LIN {X 0,Y 420.626,Z 325.953,A -85,B 0,C 180,E1 -10192.084,E2 -10192.084} C_VEL
LIN {X 0,Y 421.329,Z 314.236,A -85,B 0,C 180,E1 -10194.385,E2 -10194.385} C_VEL
LIN {X 0,Y 419.422,Z 303.683,A -85,B 0,C 180,E1 -10196.632,E2 -10196.632} C_VEL
LIN {X 0,Y 418.338,Z 298.378,A -85,B 0,C 180,E1 -10197.821,E2 -10197.821} C_VEL
LIN {X 0,Y 418.216,Z 298.389,A -85,B 0,C 180,E1 -10201.397,E2 -10201.397} C_VEL
LIN {X 0,Y 418.27,Z 298.382,A -85,B 0,C 180,E1 -10204.581,E2 -10204.581} C_VEL
LIN {X 0,Y 418.228,Z 298.387,A -85,B 0,C 180,E1 -10207.833,E2 -10207.833} C_VEL
LIN {X 0,Y 418.225,Z 298.385,A -85,B 0,C 180,E1 -10210.948,E2 -10210.948} C_VEL
LIN {X 0,Y 418.211,Z 298.387,A -85,B 0,C 180,E1 -10213.729,E2 -10213.729} C_VEL
LIN {X 0,Y 418.211,Z 298.394,A -85,B 0,C 180,E1 -10216.449,E2 -10216.449} C_VEL
LIN {X 0,Y 418.224,Z 298.386,A -85,B 0,C 180,E1 -10219.13,E2 -10219.13} C_VEL
LIN {X 0,Y 418.228,Z 298.387,A -85,B 0,C 180,E1 -10222.167,E2 -10222.167} C_VEL
LIN {X 0,Y 418.264,Z 298.38,A -85,B 0,C 180,E1 -10225.42,E2 -10225.42} C_VEL
LIN {X 0,Y 418.21,Z 298.392,A -85,B 0,C 180,E1 -10228.604,E2 -10228.604} C_VEL
LIN {X 0,Y 418.288,Z 298.376,A -85,B 0,C 180,E1 -10231.936,E2 -10231.936} C_VEL
LIN {X 0,Y 418.288,Z 298.381,A -85,B 0,C 180,E1 -10235.162,E2 -10235.162} C_VEL
LIN {X 0,Y 418.229,Z 298.385,A -85,B 0,C 180,E1 -10238.303,E2 -10238.303} C_VEL
LIN {X 0,Y 418.277,Z 298.381,A -85,B 0,C 180,E1 -10241.383,E2 -10241.383} C_VEL
LIN {X 0,Y 418.295,Z 298.376,A -85,B 0,C 180,E1 -10244.406,E2 -10244.406} C_VEL
LIN {X 0,Y 418.349,Z 298.374,A -85,B 0,C 180,E1 -10247.385,E2 -10247.385} C_VEL
LIN {X 0,Y 418.394,Z 298.371,A -85,B 0,C 180,E1 -10251.305,E2 -10251.305} C_VEL
LIN {X 0,Y 418.483,Z 298.359,A -85,B 0,C 180,E1 -10253.249,E2 -10253.249} C_VEL
LIN {X 0,Y 418.326,Z 298.377,A -85,B 0,C 180,E1 -10255.181,E2 -10255.181} C_VEL
LIN {X 0,Y 418.532,Z 298.347,A -85,B 0,C 180,E1 -10258.075,E2 -10258.075} C_VEL
LIN {X 0,Y 418.658,Z 298.332,A -85,B 0,C 180,E1 -10260,E2 -10260} C_VEL
LIN {X 0,Y 418.49,Z 298.352,A -85,B 0,C 180,E1 -10262.888,E2 -10262.888} C_VEL
LIN {X 0,Y 418.438,Z 298.358,A -85,B 0,C 180,E1 -10266.529,E2 -10266.529} C_VEL
LIN {X 0,Y 418.331,Z 298.379,A -85,B 0,C 180,E1 -10269.672,E2 -10269.672} C_VEL
LIN {X 0,Y 418.34,Z 298.37,A -85,B 0,C 180,E1 -10273,E2 -10273} C_VEL
LIN {X 0,Y 418.306,Z 298.374,A -85,B 0,C 180,E1 -10276.734,E2 -10276.734} C_VEL
LIN {X 0,Y 418.265,Z 298.385,A -85,B 0,C 180,E1 -10279.79,E2 -10279.79} C_VEL
LIN {X 0,Y 418.222,Z 298.385,A -85,B 0,C 180,E1 -10282.737,E2 -10282.737} C_VEL
LIN {X 0,Y 418.213,Z 298.391,A -85,B 0,C 180,E1 -10285.908,E2 -10285.908} C_VEL
LIN {X 0,Y 418.254,Z 298.381,A -85,B 0,C 180,E1 -10289.163,E2 -10289.163} C_VEL
LIN {X 0,Y 418.238,Z 298.387,A -85,B 0,C 180,E1 -10292.529,E2 -10292.529} C_VEL
LIN {X 0,Y 418.247,Z 298.383,A -85,B 0,C 180,E1 -10294.842,E2 -10294.842} C_VEL
LIN {X 0,Y 418.225,Z 298.392,A -85,B 0,C 180,E1 -10298.445,E2 -10298.445} C_VEL
LIN {X 0,Y 418.206,Z 298.389,A -85,B 0,C 180,E1 -10300.95,E2 -10300.95} C_VEL
LIN {X 0,Y 418.191,Z 298.389,A -85,B 0,C 180,E1 -10303.726,E2 -10303.726} C_VEL
LIN {X 0,Y 418.179,Z 298.396,A -85,B 0,C 180,E1 -10306.444,E2 -10306.444} C_VEL
LIN {X 0,Y 418.207,Z 298.389,A -85,B 0,C 180,E1 -10309.133,E2 -10309.133} C_VEL
LIN {X 0,Y 418.225,Z 298.392,A -85,B 0,C 180,E1 -10312.773,E2 -10312.773} C_VEL
LIN {X 0,Y 418.197,Z 298.39,A -85,B 0,C 180,E1 -10316.317,E2 -10316.317} C_VEL
LIN {X 0,Y 418.237,Z 298.383,A -85,B 0,C 180,E1 -10319.726,E2 -10319.726} C_VEL
LIN {X 0,Y 418.201,Z 298.395,A -85,B 0,C 180,E1 -10323.014,E2 -10323.014} C_VEL
LIN {X 0,Y 418.26,Z 298.38,A -85,B 0,C 180,E1 -10326.216,E2 -10326.216} C_VEL
LIN {X 0,Y 418.255,Z 298.386,A -85,B 0,C 180,E1 -10329.335,E2 -10329.335} C_VEL
LIN {X 0,Y 418.283,Z 298.377,A -85,B 0,C 180,E1 -10332.394,E2 -10332.394} C_VEL
LIN {X 0,Y 418.3,Z 298.381,A -85,B 0,C 180,E1 -10335.401,E2 -10335.401} C_VEL
LIN {X 0,Y 418.316,Z 298.373,A -85,B 0,C 180,E1 -10338.367,E2 -10338.367} C_VEL
LIN {X 0,Y 418.451,Z 298.356,A -85,B 0,C 180,E1 -10342.276,E2 -10342.276} C_VEL
LIN {X 0,Y 418.474,Z 298.354,A -85,B 0,C 180,E1 -10344.214,E2 -10344.214} C_VEL
LIN {X 0,Y 418.536,Z 298.348,A -85,B 0,C 180,E1 -10348.072,E2 -10348.072} C_VEL
LIN {X 0,Y 418.545,Z 298.348,A -85,B 0,C 180,E1 -10349.997,E2 -10349.997} C_VEL
LIN {X 0,Y 418.474,Z 298.353,A -85,B 0,C 180,E1 -10352.885,E2 -10352.885} C_VEL
LIN {X 0,Y 418.484,Z 298.36,A -85,B 0,C 180,E1 -10355.78,E2 -10355.78} C_VEL
LIN {X 0,Y 418.36,Z 298.372,A -85,B 0,C 180,E1 -10359.132,E2 -10359.132} C_VEL
LIN {X 0,Y 418.401,Z 298.488,A -85,B 0,C 180,E1 -10359.758,E2 -10359.758} C_VEL
LIN {X 0,Y 420.017,Z 308.097,A -85,B 0,C 180,E1 -10362.069,E2 -10362.069} C_VEL
LIN {X 0,Y 419.967,Z 311.749,A -85,B 0,C 180,E1 -10362.899,E2 -10362.899} C_VEL
LIN {X 0,Y 419.417,Z 313.02,A -85,B 0,C 180,E1 -10363.037,E2 -10363.037} C_VEL
LIN {X 0,Y 417.673,Z 315.322,A -85,B 0,C 180,E1 -10363.058,E2 -10363.058} C_VEL
LIN {X 0,Y 411.938,Z 322.29,A -85,B 0,C 180,E1 -10362.926,E2 -10362.926} C_VEL
LIN {X 0,Y 410.732,Z 325.842,A -85,B 0,C 180,E1 -10362.932,E2 -10362.932} C_VEL
LIN {X 0,Y 411.108,Z 329.038,A -85,B 0,C 180,E1 -10362.976,E2 -10362.976} C_VEL
LIN {X 0,Y 412.467,Z 332.294,A -85,B 0,C 180,E1 -10363.092,E2 -10363.092} C_VEL
LIN {X 0,Y 416.345,Z 339.616,A -85,B 0,C 180,E1 -10363.438,E2 -10363.438} C_VEL
LIN {X 0,Y 416.967,Z 343.12,A -85,B 0,C 180,E1 -10363.539,E2 -10363.539} C_VEL
LIN {X 0,Y 415.843,Z 420.461,A -85,B 0,C 180,E1 -10364.928,E2 -10364.928} C_VEL
LIN {X 0,Y 415.479,Z 434.115,A -85,B 0,C 180,E1 -10365.381,E2 -10365.381} C_VEL
LIN {X 0,Y 414.977,Z 446.178,A -85,B 0,C 180,E1 -10365.97,E2 -10365.97} C_VEL
LIN {X 0,Y 414.346,Z 458.066,A -85,B 0,C 180,E1 -10366.755,E2 -10366.755} C_VEL
LIN {X 0,Y 413.671,Z 468.928,A -85,B 0,C 180,E1 -10367.674,E2 -10367.674} C_VEL
LIN {X 0,Y 412.901,Z 478.924,A -85,B 0,C 180,E1 -10368.722,E2 -10368.722} C_VEL
LIN {X 0,Y 412.298,Z 488.255,A -85,B 0,C 180,E1 -10369.928,E2 -10369.928} C_VEL
LIN {X 0,Y 411.669,Z 496.665,A -85,B 0,C 180,E1 -10371.266,E2 -10371.266} C_VEL
LIN {X 0,Y 411.078,Z 504.603,A -85,B 0,C 180,E1 -10372.838,E2 -10372.838} C_VEL
LIN {X 0,Y 410.701,Z 510.279,A -85,B 0,C 180,E1 -10374.243,E2 -10374.243} C_VEL
LIN {X 0,Y 410.361,Z 515.517,A -85,B 0,C 180,E1 -10375.89,E2 -10375.89} C_VEL
LIN {X 0,Y 410.1,Z 519.401,A -85,B 0,C 180,E1 -10377.556,E2 -10377.556} C_VEL
LIN {X 0,Y 409.937,Z 521.797,A -85,B 0,C 180,E1 -10379.032,E2 -10379.032} C_VEL
LIN {X 0,Y 409.815,Z 523.491,A -85,B 0,C 180,E1 -10380.956,E2 -10380.956} C_VEL
LIN {X 0,Y 409.824,Z 523.714,A -85,B 0,C 180,E1 -10382.829,E2 -10382.829} C_VEL
LIN {X 0,Y 409.879,Z 522.561,A -85,B 0,C 180,E1 -10384.61,E2 -10384.61} C_VEL
LIN {X 0,Y 410.105,Z 520.141,A -85,B 0,C 180,E1 -10386.347,E2 -10386.347} C_VEL
LIN {X 0,Y 410.345,Z 516.461,A -85,B 0,C 180,E1 -10388.059,E2 -10388.059} C_VEL
LIN {X 0,Y 410.695,Z 511.796,A -85,B 0,C 180,E1 -10389.64,E2 -10389.64} C_VEL
LIN {X 0,Y 411.086,Z 505.785,A -85,B 0,C 180,E1 -10391.216,E2 -10391.216} C_VEL
LIN {X 0,Y 411.689,Z 498.204,A -85,B 0,C 180,E1 -10392.772,E2 -10392.772} C_VEL
LIN {X 0,Y 412.444,Z 489.922,A -85,B 0,C 180,E1 -10394.139,E2 -10394.139} C_VEL
LIN {X 0,Y 413.206,Z 480.472,A -85,B 0,C 180,E1 -10395.408,E2 -10395.408} C_VEL
LIN {X 0,Y 413.948,Z 469.615,A -85,B 0,C 180,E1 -10396.573,E2 -10396.573} C_VEL
LIN {X 0,Y 414.77,Z 458.24,A -85,B 0,C 180,E1 -10397.54,E2 -10397.54} C_VEL
LIN {X 0,Y 415.403,Z 446.521,A -85,B 0,C 180,E1 -10398.315,E2 -10398.315} C_VEL
LIN {X 0,Y 415.954,Z 432.986,A -85,B 0,C 180,E1 -10398.966,E2 -10398.966} C_VEL
LIN {X 0,Y 416.385,Z 419.739,A -85,B 0,C 180,E1 -10399.384,E2 -10399.384} C_VEL
LIN {X 0,Y 417.604,Z 333.211,A -85,B 0,C 180,E1 -10400.949,E2 -10400.949} C_VEL
LIN {X 0,Y 413.3,Z 312.691,A -85,B 0,C 180,E1 -10401.573,E2 -10401.573} C_VEL
LIN {X 0,Y 413.042,Z 308.119,A -85,B 0,C 180,E1 -10402.534,E2 -10402.534} C_VEL
LIN {X 0,Y 411.183,Z 299.269,A -85,B 0,C 180,E1 -10404.52,E2 -10404.52} C_VEL
LIN {X 0,Y 411.127,Z 299.276,A -85,B 0,C 180,E1 -10407.999,E2 -10407.999} C_VEL
LIN {X 0,Y 411.181,Z 299.266,A -85,B 0,C 180,E1 -10411.407,E2 -10411.407} C_VEL
LIN {X 0,Y 411.195,Z 299.268,A -85,B 0,C 180,E1 -10413.616,E2 -10413.616} C_VEL
LIN {X 0,Y 411.158,Z 299.274,A -85,B 0,C 180,E1 -10416.85,E2 -10416.85} C_VEL
LIN {X 0,Y 411.167,Z 299.271,A -85,B 0,C 180,E1 -10420.049,E2 -10420.049} C_VEL
LIN {X 0,Y 411.216,Z 299.261,A -85,B 0,C 180,E1 -10423.129,E2 -10423.129} C_VEL
LIN {X 0,Y 411.256,Z 299.258,A -85,B 0,C 180,E1 -10426.895,E2 -10426.895} C_VEL
LIN {X 0,Y 411.242,Z 299.255,A -85,B 0,C 180,E1 -10430.16,E2 -10430.16} C_VEL
LIN {X 0,Y 411.407,Z 299.237,A -85,B 0,C 180,E1 -10433.132,E2 -10433.132} C_VEL
LIN {X 0,Y 411.259,Z 299.254,A -85,B 0,C 180,E1 -10435.098,E2 -10435.098} C_VEL
LIN {X 0,Y 411.463,Z 299.228,A -85,B 0,C 180,E1 -10438.042,E2 -10438.042} C_VEL
LIN {X 0,Y 411.59,Z 299.206,A -85,B 0,C 180,E1 -10440,E2 -10440} C_VEL
LIN {X 0,Y 411.422,Z 299.234,A -85,B 0,C 180,E1 -10442.937,E2 -10442.937} C_VEL
LIN {X 0,Y 411.41,Z 299.237,A -85,B 0,C 180,E1 -10446.868,E2 -10446.868} C_VEL
LIN {X 0,Y 411.262,Z 299.254,A -85,B 0,C 180,E1 -10449.84,E2 -10449.84} C_VEL
LIN {X 0,Y 411.265,Z 299.253,A -85,B 0,C 180,E1 -10453.11,E2 -10453.11} C_VEL
LIN {X 0,Y 411.217,Z 299.255,A -85,B 0,C 180,E1 -10456.871,E2 -10456.871} C_VEL
LIN {X 0,Y 411.21,Z 299.253,A -85,B 0,C 180,E1 -10459.988,E2 -10459.988} C_VEL
LIN {X 0,Y 411.18,Z 299.267,A -85,B 0,C 180,E1 -10463.149,E2 -10463.149} C_VEL
LIN {X 0,Y 411.197,Z 299.26,A -85,B 0,C 180,E1 -10466.384,E2 -10466.384} C_VEL
LIN {X 0,Y 411.169,Z 299.268,A -85,B 0,C 180,E1 -10469.715,E2 -10469.715} C_VEL
LIN {X 0,Y 411.168,Z 299.266,A -85,B 0,C 180,E1 -10473.159,E2 -10473.159} C_VEL
LIN {X 0,Y 411.165,Z 299.266,A -85,B 0,C 180,E1 -10476.558,E2 -10476.558} C_VEL
LIN {X 0,Y 411.204,Z 299.267,A -85,B 0,C 180,E1 -10479.736,E2 -10479.736} C_VEL
LIN {X 0,Y 411.2,Z 299.266,A -85,B 0,C 180,E1 -10483.13,E2 -10483.13} C_VEL
LIN {X 0,Y 411.208,Z 299.267,A -85,B 0,C 180,E1 -10485.876,E2 -10485.876} C_VEL
LIN {X 0,Y 411.188,Z 299.27,A -85,B 0,C 180,E1 -10489.504,E2 -10489.504} C_VEL
LIN {X 0,Y 411.182,Z 299.268,A -85,B 0,C 180,E1 -10492.032,E2 -10492.032} C_VEL
LIN {X 0,Y 411.186,Z 299.271,A -85,B 0,C 180,E1 -10495.671,E2 -10495.671} C_VEL
LIN {X 0,Y 411.18,Z 299.272,A -85,B 0,C 180,E1 -10499.158,E2 -10499.158} C_VEL
LIN {X 0,Y 411.278,Z 299.342,A -85,B 0,C 180,E1 -10502.115,E2 -10502.115} C_VEL
LIN {X 0,Y 413.936,Z 312.197,A -85,B 0,C 180,E1 -10504.889,E2 -10504.889} C_VEL
LIN {X 0,Y 414.359,Z 316.233,A -85,B 0,C 180,E1 -10505.718,E2 -10505.718} C_VEL
LIN {X 0,Y 413.189,Z 333.63,A -85,B 0,C 180,E1 -10509.077,E2 -10509.077} C_VEL
LIN {X 0,Y 412.799,Z 340.804,A -85,B 0,C 180,E1 -10510.452,E2 -10510.452} C_VEL
LIN {X 0,Y 417.216,Z 368.982,A -85,B 0,C 180,E1 -10511.211,E2 -10511.211} C_VEL
LIN {X 0,Y 416.076,Z 450.173,A -85,B 0,C 180,E1 -10512.685,E2 -10512.685} C_VEL
LIN {X 0,Y 415.495,Z 463.908,A -85,B 0,C 180,E1 -10513.135,E2 -10513.135} C_VEL
LIN {X 0,Y 414.854,Z 475.762,A -85,B 0,C 180,E1 -10513.709,E2 -10513.709} C_VEL
LIN {X 0,Y 414.048,Z 487.812,A -85,B 0,C 180,E1 -10514.498,E2 -10514.498} C_VEL
LIN {X 0,Y 413.318,Z 499.293,A -85,B 0,C 180,E1 -10515.475,E2 -10515.475} C_VEL
LIN {X 0,Y 412.495,Z 509.746,A -85,B 0,C 180,E1 -10516.581,E2 -10516.581} C_VEL
LIN {X 0,Y 411.872,Z 518.266,A -85,B 0,C 180,E1 -10517.689,E2 -10517.689} C_VEL
LIN {X 0,Y 411.086,Z 527.506,A -85,B 0,C 180,E1 -10519.165,E2 -10519.165} C_VEL
LIN {X 0,Y 410.621,Z 534.957,A -85,B 0,C 180,E1 -10520.646,E2 -10520.646} C_VEL
LIN {X 0,Y 410.284,Z 540.946,A -85,B 0,C 180,E1 -10522.127,E2 -10522.127} C_VEL
LIN {X 0,Y 410.056,Z 546.105,A -85,B 0,C 180,E1 -10523.759,E2 -10523.759} C_VEL
LIN {X 0,Y 410.017,Z 549.293,A -85,B 0,C 180,E1 -10525.087,E2 -10525.087} C_VEL
LIN {X 0,Y 409.932,Z 551.145,A -85,B 0,C 180,E1 -10526.071,E2 -10526.071} C_VEL
LIN {X 0,Y 409.996,Z 553.54,A -85,B 0,C 180,E1 -10528.039,E2 -10528.039} C_VEL
LIN {X 0,Y 409.955,Z 554.143,A -85,B 0,C 180,E1 -10529.021,E2 -10529.021} C_VEL
LIN {X 0,Y 409.949,Z 554.331,A -85,B 0,C 180,E1 -10530.003,E2 -10530.003} C_VEL
LIN {X 0,Y 409.997,Z 553.467,A -85,B 0,C 180,E1 -10531.968,E2 -10531.968} C_VEL
LIN {X 0,Y 409.932,Z 552.442,A -85,B 0,C 180,E1 -10532.951,E2 -10532.951} C_VEL
LIN {X 0,Y 409.935,Z 550.987,A -85,B 0,C 180,E1 -10533.935,E2 -10533.935} C_VEL
LIN {X 0,Y 410.018,Z 547.982,A -85,B 0,C 180,E1 -10535.412,E2 -10535.412} C_VEL
LIN {X 0,Y 410.167,Z 543.911,A -85,B 0,C 180,E1 -10536.891,E2 -10536.891} C_VEL
LIN {X 0,Y 410.458,Z 537.642,A -85,B 0,C 180,E1 -10538.619,E2 -10538.619} C_VEL
LIN {X 0,Y 410.845,Z 530.811,A -85,B 0,C 180,E1 -10540.101,E2 -10540.101} C_VEL
LIN {X 0,Y 411.441,Z 522.309,A -85,B 0,C 180,E1 -10541.581,E2 -10541.581} C_VEL
LIN {X 0,Y 412.06,Z 513.546,A -85,B 0,C 180,E1 -10542.813,E2 -10542.813} C_VEL
LIN {X 0,Y 412.801,Z 503.481,A -85,B 0,C 180,E1 -10543.967,E2 -10543.967} C_VEL
LIN {X 0,Y 413.548,Z 492.018,A -85,B 0,C 180,E1 -10545.023,E2 -10545.023} C_VEL
LIN {X 0,Y 414.325,Z 479.976,A -85,B 0,C 180,E1 -10545.876,E2 -10545.876} C_VEL
LIN {X 0,Y 414.998,Z 467.447,A -85,B 0,C 180,E1 -10546.544,E2 -10546.544} C_VEL
LIN {X 0,Y 415.559,Z 454.361,A -85,B 0,C 180,E1 -10547.027,E2 -10547.027} C_VEL
LIN {X 0,Y 415.931,Z 437.009,A -85,B 0,C 180,E1 -10547.392,E2 -10547.392} C_VEL
LIN {X 0,Y 416.689,Z 368.049,A -85,B 0,C 180,E1 -10548.617,E2 -10548.617} C_VEL
LIN {X 0,Y 412.668,Z 341.785,A -85,B 0,C 180,E1 -10549.281,E2 -10549.281} C_VEL
LIN {X 0,Y 413.701,Z 325.613,A -85,B 0,C 180,E1 -10552.474,E2 -10552.474} C_VEL
LIN {X 0,Y 414.371,Z 315.206,A -85,B 0,C 180,E1 -10554.555,E2 -10554.555} C_VEL
LIN {X 0,Y 412.159,Z 303.311,A -85,B 0,C 180,E1 -10557.139,E2 -10557.139} C_VEL
LIN {X 0,Y 411.278,Z 299.257,A -85,B 0,C 180,E1 -10558.1,E2 -10558.1} C_VEL
LIN {X 0,Y 411.187,Z 299.264,A -85,B 0,C 180,E1 -10561.284,E2 -10561.284} C_VEL
LIN {X 0,Y 411.211,Z 299.264,A -85,B 0,C 180,E1 -10564.334,E2 -10564.334} C_VEL
LIN {X 0,Y 411.194,Z 299.265,A -85,B 0,C 180,E1 -10567.975,E2 -10567.975} C_VEL
LIN {X 0,Y 411.166,Z 299.264,A -85,B 0,C 180,E1 -10571.228,E2 -10571.228} C_VEL
LIN {X 0,Y 411.178,Z 299.269,A -85,B 0,C 180,E1 -10574.491,E2 -10574.491} C_VEL
LIN {X 0,Y 411.178,Z 299.266,A -85,B 0,C 180,E1 -10578.195,E2 -10578.195} C_VEL
LIN {X 0,Y 411.22,Z 299.262,A -85,B 0,C 180,E1 -10580.776,E2 -10580.776} C_VEL
LIN {X 0,Y 411.197,Z 299.265,A -85,B 0,C 180,E1 -10584.471,E2 -10584.471} C_VEL
LIN {X 0,Y 411.207,Z 299.264,A -85,B 0,C 180,E1 -10586.873,E2 -10586.873} C_VEL
LIN {X 0,Y 411.231,Z 299.262,A -85,B 0,C 180,E1 -10590.644,E2 -10590.644} C_VEL
LIN {X 0,Y 411.235,Z 299.255,A -85,B 0,C 180,E1 -10593.619,E2 -10593.619} C_VEL
LIN {X 0,Y 411.199,Z 299.266,A -85,B 0,C 180,E1 -10596.852,E2 -10596.852} C_VEL
LIN {X 0,Y 411.209,Z 299.258,A -85,B 0,C 180,E1 -10600.051,E2 -10600.051} C_VEL
LIN {X 0,Y 411.259,Z 299.259,A -85,B 0,C 180,E1 -10603.131,E2 -10603.131} C_VEL
LIN {X 0,Y 411.3,Z 299.251,A -85,B 0,C 180,E1 -10606.897,E2 -10606.897} C_VEL
LIN {X 0,Y 411.286,Z 299.249,A -85,B 0,C 180,E1 -10610.161,E2 -10610.161} C_VEL
LIN {X 0,Y 411.451,Z 299.234,A -85,B 0,C 180,E1 -10613.133,E2 -10613.133} C_VEL
LIN {X 0,Y 411.298,Z 299.252,A -85,B 0,C 180,E1 -10615.099,E2 -10615.099} C_VEL
LIN {X 0,Y 411.502,Z 299.223,A -85,B 0,C 180,E1 -10618.043,E2 -10618.043} C_VEL
LIN {X 0,Y 411.628,Z 299.208,A -85,B 0,C 180,E1 -10620,E2 -10620} C_VEL
LIN {X 0,Y 411.447,Z 299.23,A -85,B 0,C 180,E1 -10622.937,E2 -10622.937} C_VEL
LIN {X 0,Y 411.387,Z 299.236,A -85,B 0,C 180,E1 -10626.526,E2 -10626.526} C_VEL
LIN {X 0,Y 411.312,Z 299.246,A -85,B 0,C 180,E1 -10628.846,E2 -10628.846} C_VEL
LIN {X 0,Y 411.275,Z 299.257,A -85,B 0,C 180,E1 -10631.833,E2 -10631.833} C_VEL
LIN {X 0,Y 411.251,Z 299.253,A -85,B 0,C 180,E1 -10634.853,E2 -10634.853} C_VEL
LIN {X 0,Y 411.239,Z 299.263,A -85,B 0,C 180,E1 -10637.916,E2 -10637.916} C_VEL
LIN {X 0,Y 411.19,Z 299.261,A -85,B 0,C 180,E1 -10641.035,E2 -10641.035} C_VEL
LIN {X 0,Y 411.186,Z 299.267,A -85,B 0,C 180,E1 -10644.218,E2 -10644.218} C_VEL
LIN {X 0,Y 411.142,Z 299.268,A -85,B 0,C 180,E1 -10647.486,E2 -10647.486} C_VEL
LIN {X 0,Y 411.192,Z 299.263,A -85,B 0,C 180,E1 -10649.714,E2 -10649.714} C_VEL
LIN {X 0,Y 411.203,Z 299.259,A -85,B 0,C 180,E1 -10653.156,E2 -10653.156} C_VEL
LIN {X 0,Y 411.187,Z 299.266,A -85,B 0,C 180,E1 -10656.551,E2 -10656.551} C_VEL
LIN {X 0,Y 411.162,Z 299.265,A -85,B 0,C 180,E1 -10659.719,E2 -10659.719} C_VEL
LIN {X 0,Y 411.155,Z 299.266,A -85,B 0,C 180,E1 -10663.136,E2 -10663.136} C_VEL
LIN {X 0,Y 411.149,Z 299.267,A -85,B 0,C 180,E1 -10665.884,E2 -10665.884} C_VEL
LIN {X 0,Y 411.158,Z 299.265,A -85,B 0,C 180,E1 -10669.492,E2 -10669.492} C_VEL
LIN {X 0,Y 411.172,Z 299.264,A -85,B 0,C 180,E1 -10672.023,E2 -10672.023} C_VEL
LIN {X 0,Y 411.13,Z 299.272,A -85,B 0,C 180,E1 -10675.138,E2 -10675.138} C_VEL
LIN {X 0,Y 411.152,Z 299.266,A -85,B 0,C 180,E1 -10678,E2 -10678} C_VEL
LIN {X 0,Y 411.171,Z 299.265,A -85,B 0,C 180,E1 -10681.405,E2 -10681.405} C_VEL
LIN {X 0,Y 411.192,Z 299.267,A -85,B 0,C 180,E1 -10684.94,E2 -10684.94} C_VEL
LIN {X 0,Y 411.209,Z 299.259,A -85,B 0,C 180,E1 -10687.912,E2 -10687.912} C_VEL
LIN {X 0,Y 411.224,Z 299.263,A -85,B 0,C 180,E1 -10691.049,E2 -10691.049} C_VEL
LIN {X 0,Y 411.253,Z 299.253,A -85,B 0,C 180,E1 -10694.129,E2 -10694.129} C_VEL
LIN {X 0,Y 411.309,Z 299.252,A -85,B 0,C 180,E1 -10697.163,E2 -10697.163} C_VEL
LIN {X 0,Y 411.285,Z 299.249,A -85,B 0,C 180,E1 -10700.159,E2 -10700.159} C_VEL
LIN {X 0,Y 411.395,Z 299.239,A -85,B 0,C 180,E1 -10703.129,E2 -10703.129} C_VEL
LIN {X 0,Y 411.289,Z 299.251,A -85,B 0,C 180,E1 -10705.096,E2 -10705.096} C_VEL
LIN {X 0,Y 411.505,Z 299.224,A -85,B 0,C 180,E1 -10708.039,E2 -10708.039} C_VEL
LIN {X 0,Y 411.379,Z 299.238,A -85,B 0,C 180,E1 -10710.976,E2 -10710.976} C_VEL
LIN {X 0,Y 411.432,Z 299.231,A -85,B 0,C 180,E1 -10712.934,E2 -10712.934} C_VEL
LIN {X 0,Y 411.429,Z 299.239,A -85,B 0,C 180,E1 -10715.879,E2 -10715.879} C_VEL
LIN {X 0,Y 411.344,Z 299.248,A -85,B 0,C 180,E1 -10719.492,E2 -10719.492} C_VEL
LIN {X 0,Y 413.074,Z 309.584,A -85,B 0,C 180,E1 -10722.026,E2 -10722.026} C_VEL
LIN {X 0,Y 413.045,Z 313.197,A -85,B 0,C 180,E1 -10722.806,E2 -10722.806} C_VEL
LIN {X 0,Y 417.075,Z 333.227,A -85,B 0,C 180,E1 -10723.362,E2 -10723.362} C_VEL
LIN {X 0,Y 416.967,Z 343.12,A -85,B 0,C 180,E1 -10723.539,E2 -10723.539} C_VEL
LIN {X 0,Y 416.225,Z 348.959,A -85,B 0,C 180,E1 -10723.613,E2 -10723.613} C_VEL
LIN {X 0,Y 410.474,Z 367.927,A -85,B 0,C 180,E1 -10723.709,E2 -10723.709} C_VEL
LIN {X 0,Y 409.787,Z 373.763,A -85,B 0,C 180,E1 -10723.788,E2 -10723.788} C_VEL
LIN {X 0,Y 409.018,Z 421.494,A -85,B 0,C 180,E1 -10724.677,E2 -10724.677} C_VEL
LIN {X 0,Y 408.626,Z 434.931,A -85,B 0,C 180,E1 -10725.139,E2 -10725.139} C_VEL
LIN {X 0,Y 408.12,Z 446.966,A -85,B 0,C 180,E1 -10725.746,E2 -10725.746} C_VEL
LIN {X 0,Y 407.448,Z 458.565,A -85,B 0,C 180,E1 -10726.531,E2 -10726.531} C_VEL
LIN {X 0,Y 406.755,Z 469.203,A -85,B 0,C 180,E1 -10727.448,E2 -10727.448} C_VEL
LIN {X 0,Y 405.94,Z 479.466,A -85,B 0,C 180,E1 -10728.545,E2 -10728.545} C_VEL
LIN {X 0,Y 405.311,Z 488.655,A -85,B 0,C 180,E1 -10729.758,E2 -10729.758} C_VEL
LIN {X 0,Y 404.682,Z 496.881,A -85,B 0,C 180,E1 -10731.091,E2 -10731.091} C_VEL
LIN {X 0,Y 404.093,Z 503.948,A -85,B 0,C 180,E1 -10732.491,E2 -10732.491} C_VEL
LIN {X 0,Y 403.64,Z 510.619,A -85,B 0,C 180,E1 -10734.147,E2 -10734.147} C_VEL
LIN {X 0,Y 403.308,Z 515.833,A -85,B 0,C 180,E1 -10735.821,E2 -10735.821} C_VEL
LIN {X 0,Y 403.053,Z 519.108,A -85,B 0,C 180,E1 -10737.216,E2 -10737.216} C_VEL
LIN {X 0,Y 402.931,Z 520.732,A -85,B 0,C 180,E1 -10738.089,E2 -10738.089} C_VEL
LIN {X 0,Y 402.818,Z 522.366,A -85,B 0,C 180,E1 -10739.266,E2 -10739.266} C_VEL
LIN {X 0,Y 402.734,Z 523.892,A -85,B 0,C 180,E1 -10741.23,E2 -10741.23} C_VEL
LIN {X 0,Y 402.74,Z 523.889,A -85,B 0,C 180,E1 -10743.11,E2 -10743.11} C_VEL
LIN {X 0,Y 402.844,Z 522.306,A -85,B 0,C 180,E1 -10745.143,E2 -10745.143} C_VEL
LIN {X 0,Y 403.103,Z 519.984,A -85,B 0,C 180,E1 -10746.678,E2 -10746.678} C_VEL
LIN {X 0,Y 403.314,Z 516.297,A -85,B 0,C 180,E1 -10748.357,E2 -10748.357} C_VEL
LIN {X 0,Y 403.698,Z 511.031,A -85,B 0,C 180,E1 -10750.093,E2 -10750.093} C_VEL
LIN {X 0,Y 404.259,Z 504.208,A -85,B 0,C 180,E1 -10751.807,E2 -10751.807} C_VEL
LIN {X 0,Y 404.827,Z 497.332,A -85,B 0,C 180,E1 -10753.185,E2 -10753.185} C_VEL
LIN {X 0,Y 405.611,Z 489.18,A -85,B 0,C 180,E1 -10754.518,E2 -10754.518} C_VEL
LIN {X 0,Y 406.46,Z 479.11,A -85,B 0,C 180,E1 -10755.845,E2 -10755.845} C_VEL
LIN {X 0,Y 407.208,Z 468.328,A -85,B 0,C 180,E1 -10756.991,E2 -10756.991} C_VEL
LIN {X 0,Y 408.07,Z 456.749,A -85,B 0,C 180,E1 -10757.955,E2 -10757.955} C_VEL
LIN {X 0,Y 408.726,Z 445.42,A -85,B 0,C 180,E1 -10758.685,E2 -10758.685} C_VEL
LIN {X 0,Y 409.272,Z 432.759,A -85,B 0,C 180,E1 -10759.291,E2 -10759.291} C_VEL
LIN {X 0,Y 409.636,Z 420.718,A -85,B 0,C 180,E1 -10759.68,E2 -10759.68} C_VEL
LIN {X 0,Y 410.945,Z 334.122,A -85,B 0,C 180,E1 -10761.277,E2 -10761.277} C_VEL
LIN {X 0,Y 406.47,Z 312.965,A -85,B 0,C 180,E1 -10761.938,E2 -10761.938} C_VEL
LIN {X 0,Y 405.87,Z 308.289,A -85,B 0,C 180,E1 -10762.959,E2 -10762.959} C_VEL
LIN {X 0,Y 404.139,Z 300.147,A -85,B 0,C 180,E1 -10764.807,E2 -10764.807} C_VEL
LIN {X 0,Y 404.103,Z 300.148,A -85,B 0,C 180,E1 -10767.375,E2 -10767.375} C_VEL
LIN {X 0,Y 404.142,Z 300.145,A -85,B 0,C 180,E1 -10770.862,E2 -10770.862} C_VEL
LIN {X 0,Y 404.153,Z 300.145,A -85,B 0,C 180,E1 -10773.12,E2 -10773.12} C_VEL
LIN {X 0,Y 404.133,Z 300.148,A -85,B 0,C 180,E1 -10775.331,E2 -10775.331} C_VEL
LIN {X 0,Y 404.092,Z 300.154,A -85,B 0,C 180,E1 -10778.578,E2 -10778.578} C_VEL
LIN {X 0,Y 404.161,Z 300.139,A -85,B 0,C 180,E1 -10781.76,E2 -10781.76} C_VEL
LIN {X 0,Y 404.156,Z 300.143,A -85,B 0,C 180,E1 -10784.88,E2 -10784.88} C_VEL
LIN {X 0,Y 404.206,Z 300.133,A -85,B 0,C 180,E1 -10787.957,E2 -10787.957} C_VEL
LIN {X 0,Y 404.356,Z 300.114,A -85,B 0,C 180,E1 -10792.127,E2 -10792.127} C_VEL
LIN {X 0,Y 404.369,Z 300.112,A -85,B 0,C 180,E1 -10794.014,E2 -10794.014} C_VEL
LIN {X 0,Y 404.432,Z 300.104,A -85,B 0,C 180,E1 -10798.008,E2 -10798.008} C_VEL
LIN {X 0,Y 404.56,Z 300.082,A -85,B 0,C 180,E1 -10800,E2 -10800} C_VEL
LIN {X 0,Y 404.379,Z 300.11,A -85,B 0,C 180,E1 -10802.989,E2 -10802.989} C_VEL
LIN {X 0,Y 404.357,Z 300.114,A -85,B 0,C 180,E1 -10806.988,E2 -10806.988} C_VEL
LIN {X 0,Y 404.224,Z 300.13,A -85,B 0,C 180,E1 -10810.013,E2 -10810.013} C_VEL
LIN {X 0,Y 404.218,Z 300.132,A -85,B 0,C 180,E1 -10813.213,E2 -10813.213} C_VEL
LIN {X 0,Y 404.171,Z 300.134,A -85,B 0,C 180,E1 -10817.01,E2 -10817.01} C_VEL
LIN {X 0,Y 404.161,Z 300.131,A -85,B 0,C 180,E1 -10820.352,E2 -10820.352} C_VEL
LIN {X 0,Y 404.138,Z 300.137,A -85,B 0,C 180,E1 -10823.577,E2 -10823.577} C_VEL
LIN {X 0,Y 404.154,Z 300.139,A -85,B 0,C 180,E1 -10826.88,E2 -10826.88} C_VEL
LIN {X 0,Y 404.113,Z 300.143,A -85,B 0,C 180,E1 -10830.288,E2 -10830.288} C_VEL
LIN {X 0,Y 404.107,Z 300.147,A -85,B 0,C 180,E1 -10833.816,E2 -10833.816} C_VEL
LIN {X 0,Y 404.116,Z 300.145,A -85,B 0,C 180,E1 -10836.882,E2 -10836.882} C_VEL
LIN {X 0,Y 404.142,Z 300.144,A -85,B 0,C 180,E1 -10840.048,E2 -10840.048} C_VEL
LIN {X 0,Y 404.174,Z 300.141,A -85,B 0,C 180,E1 -10843.096,E2 -10843.096} C_VEL
LIN {X 0,Y 404.181,Z 300.142,A -85,B 0,C 180,E1 -10845.939,E2 -10845.939} C_VEL
LIN {X 0,Y 404.138,Z 300.144,A -85,B 0,C 180,E1 -10848.645,E2 -10848.645} C_VEL
LIN {X 0,Y 404.139,Z 300.146,A -85,B 0,C 180,E1 -10851.495,E2 -10851.495} C_VEL
LIN {X 0,Y 404.164,Z 300.141,A -85,B 0,C 180,E1 -10854.989,E2 -10854.989} C_VEL
LIN {X 0,Y 404.128,Z 300.149,A -85,B 0,C 180,E1 -10858.559,E2 -10858.559} C_VEL
LIN {X 0,Y 404.229,Z 300.19,A -85,B 0,C 180,E1 -10861.797,E2 -10861.797} C_VEL
LIN {X 0,Y 406.987,Z 313.375,A -85,B 0,C 180,E1 -10864.703,E2 -10864.703} C_VEL
LIN {X 0,Y 407.458,Z 317.411,A -85,B 0,C 180,E1 -10865.551,E2 -10865.551} C_VEL
LIN {X 0,Y 406.327,Z 333.455,A -85,B 0,C 180,E1 -10868.707,E2 -10868.707} C_VEL
LIN {X 0,Y 405.928,Z 340.48,A -85,B 0,C 180,E1 -10870.079,E2 -10870.079} C_VEL
LIN {X 0,Y 410.444,Z 368.958,A -85,B 0,C 180,E1 -10870.871,E2 -10870.871} C_VEL
LIN {X 0,Y 409.382,Z 448.116,A -85,B 0,C 180,E1 -10872.328,E2 -10872.328} C_VEL
LIN {X 0,Y 408.894,Z 461.002,A -85,B 0,C 180,E1 -10872.725,E2 -10872.725} C_VEL
LIN {X 0,Y 408.196,Z 473.511,A -85,B 0,C 180,E1 -10873.307,E2 -10873.307} C_VEL
LIN {X 0,Y 407.334,Z 486.104,A -85,B 0,C 180,E1 -10874.108,E2 -10874.108} C_VEL
LIN {X 0,Y 406.494,Z 498.031,A -85,B 0,C 180,E1 -10875.115,E2 -10875.115} C_VEL
LIN {X 0,Y 405.698,Z 508.51,A -85,B 0,C 180,E1 -10876.224,E2 -10876.224} C_VEL
LIN {X 0,Y 404.916,Z 518.086,A -85,B 0,C 180,E1 -10877.474,E2 -10877.474} C_VEL
LIN {X 0,Y 404.084,Z 527.308,A -85,B 0,C 180,E1 -10878.974,E2 -10878.974} C_VEL
LIN {X 0,Y 403.599,Z 534.75,A -85,B 0,C 180,E1 -10880.482,E2 -10880.482} C_VEL
LIN {X 0,Y 403.215,Z 540.728,A -85,B 0,C 180,E1 -10881.988,E2 -10881.988} C_VEL
LIN {X 0,Y 402.976,Z 546.184,A -85,B 0,C 180,E1 -10883.771,E2 -10883.771} C_VEL
LIN {X 0,Y 402.929,Z 549.058,A -85,B 0,C 180,E1 -10885,E2 -10885} C_VEL
LIN {X 0,Y 402.853,Z 550.9,A -85,B 0,C 180,E1 -10886.002,E2 -10886.002} C_VEL
LIN {X 0,Y 402.906,Z 553.286,A -85,B 0,C 180,E1 -10888.004,E2 -10888.004} C_VEL
LIN {X 0,Y 402.882,Z 553.886,A -85,B 0,C 180,E1 -10889.004,E2 -10889.004} C_VEL
LIN {X 0,Y 402.873,Z 554.064,A -85,B 0,C 180,E1 -10890.003,E2 -10890.003} C_VEL
LIN {X 0,Y 402.882,Z 553.821,A -85,B 0,C 180,E1 -10891.003,E2 -10891.003} C_VEL
LIN {X 0,Y 402.907,Z 553.188,A -85,B 0,C 180,E1 -10892.002,E2 -10892.002} C_VEL
LIN {X 0,Y 402.833,Z 552.157,A -85,B 0,C 180,E1 -10893.003,E2 -10893.003} C_VEL
LIN {X 0,Y 402.855,Z 550.69,A -85,B 0,C 180,E1 -10894.004,E2 -10894.004} C_VEL
LIN {X 0,Y 402.916,Z 547.671,A -85,B 0,C 180,E1 -10895.508,E2 -10895.508} C_VEL
LIN {X 0,Y 403.079,Z 543.585,A -85,B 0,C 180,E1 -10897.013,E2 -10897.013} C_VEL
LIN {X 0,Y 403.393,Z 537.298,A -85,B 0,C 180,E1 -10898.771,E2 -10898.771} C_VEL
LIN {X 0,Y 403.798,Z 530.446,A -85,B 0,C 180,E1 -10900.279,E2 -10900.279} C_VEL
LIN {X 0,Y 404.444,Z 521.911,A -85,B 0,C 180,E1 -10901.784,E2 -10901.784} C_VEL
LIN {X 0,Y 405.086,Z 513.119,A -85,B 0,C 180,E1 -10903.037,E2 -10903.037} C_VEL
LIN {X 0,Y 405.907,Z 502.54,A -85,B 0,C 180,E1 -10904.261,E2 -10904.261} C_VEL
LIN {X 0,Y 406.671,Z 491.496,A -85,B 0,C 180,E1 -10905.283,E2 -10905.283} C_VEL
LIN {X 0,Y 407.45,Z 479.373,A -85,B 0,C 180,E1 -10906.151,E2 -10906.151} C_VEL
LIN {X 0,Y 408.194,Z 466.747,A -85,B 0,C 180,E1 -10906.828,E2 -10906.828} C_VEL
LIN {X 0,Y 408.718,Z 454.461,A -85,B 0,C 180,E1 -10907.289,E2 -10907.289} C_VEL
LIN {X 0,Y 409.1,Z 439.063,A -85,B 0,C 180,E1 -10907.627,E2 -10907.627} C_VEL
LIN {X 0,Y 409.869,Z 368.663,A -85,B 0,C 180,E1 -10908.902,E2 -10908.902} C_VEL
LIN {X 0,Y 405.755,Z 341.375,A -85,B 0,C 180,E1 -10909.636,E2 -10909.636} C_VEL
LIN {X 0,Y 406.847,Z 325.267,A -85,B 0,C 180,E1 -10912.874,E2 -10912.874} C_VEL
LIN {X 0,Y 407.39,Z 316.147,A -85,B 0,C 180,E1 -10914.732,E2 -10914.732} C_VEL
LIN {X 0,Y 405.199,Z 304.587,A -85,B 0,C 180,E1 -10917.296,E2 -10917.296} C_VEL
LIN {X 0,Y 404.225,Z 300.134,A -85,B 0,C 180,E1 -10918.352,E2 -10918.352} C_VEL
LIN {X 0,Y 404.144,Z 300.142,A -85,B 0,C 180,E1 -10921.559,E2 -10921.559} C_VEL
LIN {X 0,Y 404.189,Z 300.133,A -85,B 0,C 180,E1 -10925.017,E2 -10925.017} C_VEL
LIN {X 0,Y 404.152,Z 300.139,A -85,B 0,C 180,E1 -10928.758,E2 -10928.758} C_VEL
LIN {X 0,Y 404.125,Z 300.141,A -85,B 0,C 180,E1 -10931.6,E2 -10931.6} C_VEL
LIN {X 0,Y 404.147,Z 300.144,A -85,B 0,C 180,E1 -10934.522,E2 -10934.522} C_VEL
LIN {X 0,Y 404.137,Z 300.139,A -85,B 0,C 180,E1 -10937.296,E2 -10937.296} C_VEL
LIN {X 0,Y 404.171,Z 300.137,A -85,B 0,C 180,E1 -10939.955,E2 -10939.955} C_VEL
LIN {X 0,Y 404.136,Z 300.141,A -85,B 0,C 180,E1 -10943.125,E2 -10943.125} C_VEL
LIN {X 0,Y 404.144,Z 300.14,A -85,B 0,C 180,E1 -10946.188,E2 -10946.188} C_VEL
LIN {X 0,Y 404.144,Z 300.138,A -85,B 0,C 180,E1 -10949.715,E2 -10949.715} C_VEL
LIN {X 0,Y 404.193,Z 300.137,A -85,B 0,C 180,E1 -10953.123,E2 -10953.123} C_VEL
LIN {X 0,Y 404.174,Z 300.137,A -85,B 0,C 180,E1 -10955.334,E2 -10955.334} C_VEL
LIN {X 0,Y 404.134,Z 300.143,A -85,B 0,C 180,E1 -10958.58,E2 -10958.58} C_VEL
LIN {X 0,Y 404.205,Z 300.132,A -85,B 0,C 180,E1 -10961.762,E2 -10961.762} C_VEL
LIN {X 0,Y 404.199,Z 300.136,A -85,B 0,C 180,E1 -10964.882,E2 -10964.882} C_VEL
LIN {X 0,Y 404.25,Z 300.126,A -85,B 0,C 180,E1 -10967.958,E2 -10967.958} C_VEL
LIN {X 0,Y 404.402,Z 300.107,A -85,B 0,C 180,E1 -10972.128,E2 -10972.128} C_VEL
LIN {X 0,Y 404.412,Z 300.106,A -85,B 0,C 180,E1 -10974.015,E2 -10974.015} C_VEL
LIN {X 0,Y 404.471,Z 300.099,A -85,B 0,C 180,E1 -10978.009,E2 -10978.009} C_VEL
LIN {X 0,Y 404.598,Z 300.084,A -85,B 0,C 180,E1 -10980,E2 -10980} C_VEL
LIN {X 0,Y 404.405,Z 300.107,A -85,B 0,C 180,E1 -10982.989,E2 -10982.989} C_VEL
LIN {X 0,Y 404.339,Z 300.114,A -85,B 0,C 180,E1 -10986.521,E2 -10986.521} C_VEL
LIN {X 0,Y 404.259,Z 300.125,A -85,B 0,C 180,E1 -10989.002,E2 -10989.002} C_VEL
LIN {X 0,Y 404.249,Z 300.13,A -85,B 0,C 180,E1 -10992.042,E2 -10992.042} C_VEL
LIN {X 0,Y 404.198,Z 300.132,A -85,B 0,C 180,E1 -10995.118,E2 -10995.118} C_VEL
LIN {X 0,Y 404.198,Z 300.135,A -85,B 0,C 180,E1 -10998.239,E2 -10998.239} C_VEL
LIN {X 0,Y 404.132,Z 300.141,A -85,B 0,C 180,E1 -11001.42,E2 -11001.42} C_VEL
LIN {X 0,Y 404.132,Z 300.141,A -85,B 0,C 180,E1 -11004.669,E2 -11004.669} C_VEL
LIN {X 0,Y 404.1,Z 300.15,A -85,B 0,C 180,E1 -11008.007,E2 -11008.007} C_VEL
LIN {X 0,Y 404.14,Z 300.146,A -85,B 0,C 180,E1 -11010.286,E2 -11010.286} C_VEL
LIN {X 0,Y 404.136,Z 300.142,A -85,B 0,C 180,E1 -11013.813,E2 -11013.813} C_VEL
LIN {X 0,Y 404.129,Z 300.142,A -85,B 0,C 180,E1 -11016.873,E2 -11016.873} C_VEL
LIN {X 0,Y 404.118,Z 300.145,A -85,B 0,C 180,E1 -11020.075,E2 -11020.075} C_VEL
LIN {X 0,Y 404.136,Z 300.141,A -85,B 0,C 180,E1 -11023.081,E2 -11023.081} C_VEL
LIN {X 0,Y 404.107,Z 300.144,A -85,B 0,C 180,E1 -11025.92,E2 -11025.92} C_VEL
LIN {X 0,Y 404.1,Z 300.152,A -85,B 0,C 180,E1 -11028.632,E2 -11028.632} C_VEL
LIN {X 0,Y 404.13,Z 300.141,A -85,B 0,C 180,E1 -11031.497,E2 -11031.497} C_VEL
LIN {X 0,Y 404.089,Z 300.151,A -85,B 0,C 180,E1 -11034.973,E2 -11034.973} C_VEL
LIN {X 0,Y 404.132,Z 300.143,A -85,B 0,C 180,E1 -11038.444,E2 -11038.444} C_VEL
LIN {X 0,Y 404.151,Z 300.144,A -85,B 0,C 180,E1 -11040.861,E2 -11040.861} C_VEL
LIN {X 0,Y 404.156,Z 300.141,A -85,B 0,C 180,E1 -11044.722,E2 -11044.722} C_VEL
LIN {X 0,Y 404.172,Z 300.138,A -85,B 0,C 180,E1 -11047.506,E2 -11047.506} C_VEL
LIN {X 0,Y 404.168,Z 300.138,A -85,B 0,C 180,E1 -11050.706,E2 -11050.706} C_VEL
LIN {X 0,Y 404.222,Z 300.13,A -85,B 0,C 180,E1 -11053.846,E2 -11053.846} C_VEL
LIN {X 0,Y 404.289,Z 300.123,A -85,B 0,C 180,E1 -11056.937,E2 -11056.937} C_VEL
LIN {X 0,Y 404.253,Z 300.126,A -85,B 0,C 180,E1 -11059.986,E2 -11059.986} C_VEL
LIN {X 0,Y 404.345,Z 300.116,A -85,B 0,C 180,E1 -11063.009,E2 -11063.009} C_VEL
LIN {X 0,Y 404.261,Z 300.126,A -85,B 0,C 180,E1 -11065.01,E2 -11065.01} C_VEL
LIN {X 0,Y 404.473,Z 300.1,A -85,B 0,C 180,E1 -11068.005,E2 -11068.005} C_VEL
LIN {X 0,Y 404.349,Z 300.114,A -85,B 0,C 180,E1 -11070.993,E2 -11070.993} C_VEL
LIN {X 0,Y 404.392,Z 300.108,A -85,B 0,C 180,E1 -11072.985,E2 -11072.985} C_VEL
LIN {X 0,Y 404.377,Z 300.117,A -85,B 0,C 180,E1 -11075.982,E2 -11075.982} C_VEL
LIN {X 0,Y 404.33,Z 300.273,A -85,B 0,C 180,E1 -11079.311,E2 -11079.311} C_VEL
LIN {X 0,Y 406.088,Z 309.981,A -85,B 0,C 180,E1 -11081.729,E2 -11081.729} C_VEL
LIN {X 0,Y 406.088,Z 313.082,A -85,B 0,C 180,E1 -11082.458,E2 -11082.458} C_VEL
LIN {X 0,Y 410.324,Z 334.529,A -85,B 0,C 180,E1 -11083.082,E2 -11083.082} C_VEL
LIN {X 0,Y 409.787,Z 373.763,A -85,B 0,C 180,E1 -11083.788,E2 -11083.788} C_VEL
LIN {X 0,Y 409.094,Z 379.601,A -85,B 0,C 180,E1 -11083.866,E2 -11083.866} C_VEL
LIN {X 0,Y 403.28,Z 398.56,A -85,B 0,C 180,E1 -11083.968,E2 -11083.968} C_VEL
LIN {X 0,Y 402.524,Z 404.4,A -85,B 0,C 180,E1 -11084.046,E2 -11084.046} C_VEL
LIN {X 0,Y 402.156,Z 423.636,A -85,B 0,C 180,E1 -11084.448,E2 -11084.448} C_VEL
LIN {X 0,Y 401.782,Z 435.611,A -85,B 0,C 180,E1 -11084.883,E2 -11084.883} C_VEL
LIN {X 0,Y 401.219,Z 448.237,A -85,B 0,C 180,E1 -11085.546,E2 -11085.546} C_VEL
LIN {X 0,Y 400.475,Z 460.736,A -85,B 0,C 180,E1 -11086.434,E2 -11086.434} C_VEL
LIN {X 0,Y 399.75,Z 471.217,A -85,B 0,C 180,E1 -11087.385,E2 -11087.385} C_VEL
LIN {X 0,Y 398.929,Z 481.008,A -85,B 0,C 180,E1 -11088.483,E2 -11088.483} C_VEL
LIN {X 0,Y 398.144,Z 490.848,A -85,B 0,C 180,E1 -11089.859,E2 -11089.859} C_VEL
LIN {X 0,Y 397.569,Z 498.869,A -85,B 0,C 180,E1 -11091.242,E2 -11091.242} C_VEL
LIN {X 0,Y 397.012,Z 505.514,A -85,B 0,C 180,E1 -11092.64,E2 -11092.64} C_VEL
LIN {X 0,Y 396.593,Z 510.954,A -85,B 0,C 180,E1 -11094.048,E2 -11094.048} C_VEL
LIN {X 0,Y 396.24,Z 516.151,A -85,B 0,C 180,E1 -11095.751,E2 -11095.751} C_VEL
LIN {X 0,Y 395.914,Z 520.009,A -85,B 0,C 180,E1 -11097.48,E2 -11097.48} C_VEL
LIN {X 0,Y 395.718,Z 522.94,A -85,B 0,C 180,E1 -11099.512,E2 -11099.512} C_VEL
LIN {X 0,Y 395.637,Z 524.235,A -85,B 0,C 180,E1 -11101.497,E2 -11101.497} C_VEL
LIN {X 0,Y 395.64,Z 524.038,A -85,B 0,C 180,E1 -11103.407,E2 -11103.407} C_VEL
LIN {X 0,Y 395.782,Z 522.556,A -85,B 0,C 180,E1 -11105.231,E2 -11105.231} C_VEL
LIN {X 0,Y 396.06,Z 519.662,A -85,B 0,C 180,E1 -11107.101,E2 -11107.101} C_VEL
LIN {X 0,Y 396.328,Z 515.954,A -85,B 0,C 180,E1 -11108.717,E2 -11108.717} C_VEL
LIN {X 0,Y 396.701,Z 510.867,A -85,B 0,C 180,E1 -11110.377,E2 -11110.377} C_VEL
LIN {X 0,Y 397.276,Z 504.421,A -85,B 0,C 180,E1 -11112.012,E2 -11112.012} C_VEL
LIN {X 0,Y 397.993,Z 496.443,A -85,B 0,C 180,E1 -11113.614,E2 -11113.614} C_VEL
LIN {X 0,Y 398.837,Z 487.697,A -85,B 0,C 180,E1 -11115.012,E2 -11115.012} C_VEL
LIN {X 0,Y 399.718,Z 477.876,A -85,B 0,C 180,E1 -11116.287,E2 -11116.287} C_VEL
LIN {X 0,Y 400.462,Z 467.677,A -85,B 0,C 180,E1 -11117.361,E2 -11117.361} C_VEL
LIN {X 0,Y 401.319,Z 456.586,A -85,B 0,C 180,E1 -11118.282,E2 -11118.282} C_VEL
LIN {X 0,Y 401.996,Z 445.23,A -85,B 0,C 180,E1 -11119.019,E2 -11119.019} C_VEL
LIN {X 0,Y 402.589,Z 432.37,A -85,B 0,C 180,E1 -11119.635,E2 -11119.635} C_VEL
LIN {X 0,Y 402.982,Z 419.204,A -85,B 0,C 180,E1 -11120.044,E2 -11120.044} C_VEL
LIN {X 0,Y 404.238,Z 334.732,A -85,B 0,C 180,E1 -11121.626,E2 -11121.626} C_VEL
LIN {X 0,Y 399.693,Z 313.811,A -85,B 0,C 180,E1 -11122.298,E2 -11122.298} C_VEL
LIN {X 0,Y 399.571,Z 313.3,A -85,B 0,C 180,E1 -11122.315,E2 -11122.315} C_VEL
LIN {X 0,Y 397.175,Z 301.333,A -85,B 0,C 180,E1 -11125.049,E2 -11125.049} C_VEL
LIN {X 0,Y 397.102,Z 301.022,A -85,B 0,C 180,E1 -11125.196,E2 -11125.196} C_VEL
LIN {X 0,Y 397.045,Z 301.03,A -85,B 0,C 180,E1 -11128.16,E2 -11128.16} C_VEL
LIN {X 0,Y 397.085,Z 301.022,A -85,B 0,C 180,E1 -11131.453,E2 -11131.453} C_VEL
LIN {X 0,Y 397.11,Z 301.025,A -85,B 0,C 180,E1 -11134.485,E2 -11134.485} C_VEL
LIN {X 0,Y 397.064,Z 301.029,A -85,B 0,C 180,E1 -11137.083,E2 -11137.083} C_VEL
LIN {X 0,Y 397.101,Z 301.027,A -85,B 0,C 180,E1 -11140.35,E2 -11140.35} C_VEL
LIN {X 0,Y 397.118,Z 301.015,A -85,B 0,C 180,E1 -11143.551,E2 -11143.551} C_VEL
LIN {X 0,Y 397.181,Z 301.01,A -85,B 0,C 180,E1 -11146.701,E2 -11146.701} C_VEL
LIN {X 0,Y 397.168,Z 301.006,A -85,B 0,C 180,E1 -11149.808,E2 -11149.808} C_VEL
LIN {X 0,Y 397.304,Z 300.993,A -85,B 0,C 180,E1 -11152.887,E2 -11152.887} C_VEL
LIN {X 0,Y 397.203,Z 301.006,A -85,B 0,C 180,E1 -11154.924,E2 -11154.924} C_VEL
LIN {X 0,Y 397.402,Z 300.98,A -85,B 0,C 180,E1 -11157.973,E2 -11157.973} C_VEL
LIN {X 0,Y 397.529,Z 300.957,A -85,B 0,C 180,E1 -11160,E2 -11160} C_VEL
LIN {X 0,Y 397.338,Z 300.986,A -85,B 0,C 180,E1 -11163.042,E2 -11163.042} C_VEL
LIN {X 0,Y 397.326,Z 300.989,A -85,B 0,C 180,E1 -11166.092,E2 -11166.092} C_VEL
LIN {X 0,Y 397.21,Z 301.007,A -85,B 0,C 180,E1 -11169.163,E2 -11169.163} C_VEL
LIN {X 0,Y 397.182,Z 301,A -85,B 0,C 180,E1 -11172.259,E2 -11172.259} C_VEL
LIN {X 0,Y 397.137,Z 301.011,A -85,B 0,C 180,E1 -11175.394,E2 -11175.394} C_VEL
LIN {X 0,Y 397.125,Z 301.013,A -85,B 0,C 180,E1 -11178.575,E2 -11178.575} C_VEL
LIN {X 0,Y 397.123,Z 301.014,A -85,B 0,C 180,E1 -11181.817,E2 -11181.817} C_VEL
LIN {X 0,Y 397.111,Z 301.017,A -85,B 0,C 180,E1 -11185.515,E2 -11185.515} C_VEL
LIN {X 0,Y 397.085,Z 301.013,A -85,B 0,C 180,E1 -11188.547,E2 -11188.547} C_VEL
LIN {X 0,Y 397.041,Z 301.024,A -85,B 0,C 180,E1 -11192.075,E2 -11192.075} C_VEL
LIN {X 0,Y 397.084,Z 301.021,A -85,B 0,C 180,E1 -11195.507,E2 -11195.507} C_VEL
LIN {X 0,Y 397.14,Z 301.012,A -85,B 0,C 180,E1 -11198.873,E2 -11198.873} C_VEL
LIN {X 0,Y 397.129,Z 301.019,A -85,B 0,C 180,E1 -11202.259,E2 -11202.259} C_VEL
LIN {X 0,Y 397.122,Z 301.02,A -85,B 0,C 180,E1 -11205.064,E2 -11205.064} C_VEL
LIN {X 0,Y 397.129,Z 301.02,A -85,B 0,C 180,E1 -11208.011,E2 -11208.011} C_VEL
LIN {X 0,Y 397.087,Z 301.024,A -85,B 0,C 180,E1 -11211.731,E2 -11211.731} C_VEL
LIN {X 0,Y 397.105,Z 301.024,A -85,B 0,C 180,E1 -11215.511,E2 -11215.511} C_VEL
LIN {X 0,Y 397.067,Z 301.03,A -85,B 0,C 180,E1 -11219.123,E2 -11219.123} C_VEL
LIN {X 0,Y 397.171,Z 301.038,A -85,B 0,C 180,E1 -11221.466,E2 -11221.466} C_VEL
LIN {X 0,Y 400.036,Z 314.55,A -85,B 0,C 180,E1 -11224.511,E2 -11224.511} C_VEL
LIN {X 0,Y 400.546,Z 318.428,A -85,B 0,C 180,E1 -11225.345,E2 -11225.345} C_VEL
LIN {X 0,Y 399.487,Z 333.305,A -85,B 0,C 180,E1 -11228.324,E2 -11228.324} C_VEL
LIN {X 0,Y 399.031,Z 340.175,A -85,B 0,C 180,E1 -11229.688,E2 -11229.688} C_VEL
LIN {X 0,Y 403.145,Z 365.477,A -85,B 0,C 180,E1 -11230.424,E2 -11230.424} C_VEL
LIN {X 0,Y 403.872,Z 370.604,A -85,B 0,C 180,E1 -11230.562,E2 -11230.562} C_VEL
LIN {X 0,Y 402.629,Z 449.827,A -85,B 0,C 180,E1 -11232.054,E2 -11232.054} C_VEL
LIN {X 0,Y 401.99,Z 463.466,A -85,B 0,C 180,E1 -11232.518,E2 -11232.518} C_VEL
LIN {X 0,Y 401.246,Z 475.813,A -85,B 0,C 180,E1 -11233.141,E2 -11233.141} C_VEL
LIN {X 0,Y 400.394,Z 487.684,A -85,B 0,C 180,E1 -11233.956,E2 -11233.956} C_VEL
LIN {X 0,Y 399.515,Z 499.381,A -85,B 0,C 180,E1 -11234.992,E2 -11234.992} C_VEL
LIN {X 0,Y 398.702,Z 509.348,A -85,B 0,C 180,E1 -11236.094,E2 -11236.094} C_VEL
LIN {X 0,Y 397.967,Z 517.926,A -85,B 0,C 180,E1 -11237.251,E2 -11237.251} C_VEL
LIN {X 0,Y 397.082,Z 527.118,A -85,B 0,C 180,E1 -11238.778,E2 -11238.778} C_VEL
LIN {X 0,Y 396.556,Z 534.541,A -85,B 0,C 180,E1 -11240.311,E2 -11240.311} C_VEL
LIN {X 0,Y 396.169,Z 540.51,A -85,B 0,C 180,E1 -11241.845,E2 -11241.845} C_VEL
LIN {X 0,Y 395.934,Z 545.226,A -85,B 0,C 180,E1 -11243.379,E2 -11243.379} C_VEL
LIN {X 0,Y 395.843,Z 548.823,A -85,B 0,C 180,E1 -11244.911,E2 -11244.911} C_VEL
LIN {X 0,Y 395.775,Z 550.655,A -85,B 0,C 180,E1 -11245.93,E2 -11245.93} C_VEL
LIN {X 0,Y 395.804,Z 553.033,A -85,B 0,C 180,E1 -11247.968,E2 -11247.968} C_VEL
LIN {X 0,Y 395.81,Z 553.63,A -85,B 0,C 180,E1 -11248.986,E2 -11248.986} C_VEL
LIN {X 0,Y 395.799,Z 553.796,A -85,B 0,C 180,E1 -11250.003,E2 -11250.003} C_VEL
LIN {X 0,Y 395.81,Z 553.548,A -85,B 0,C 180,E1 -11251.021,E2 -11251.021} C_VEL
LIN {X 0,Y 395.805,Z 552.909,A -85,B 0,C 180,E1 -11252.038,E2 -11252.038} C_VEL
LIN {X 0,Y 395.735,Z 551.872,A -85,B 0,C 180,E1 -11253.057,E2 -11253.057} C_VEL
LIN {X 0,Y 395.778,Z 550.393,A -85,B 0,C 180,E1 -11254.076,E2 -11254.076} C_VEL
LIN {X 0,Y 395.828,Z 546.868,A -85,B 0,C 180,E1 -11255.807,E2 -11255.807} C_VEL
LIN {X 0,Y 396.066,Z 541.627,A -85,B 0,C 180,E1 -11257.651,E2 -11257.651} C_VEL
LIN {X 0,Y 396.449,Z 534.832,A -85,B 0,C 180,E1 -11259.441,E2 -11259.441} C_VEL
LIN {X 0,Y 396.946,Z 527.418,A -85,B 0,C 180,E1 -11260.975,E2 -11260.975} C_VEL
LIN {X 0,Y 397.764,Z 518.217,A -85,B 0,C 180,E1 -11262.503,E2 -11262.503} C_VEL
LIN {X 0,Y 398.526,Z 508.108,A -85,B 0,C 180,E1 -11263.839,E2 -11263.839} C_VEL
LIN {X 0,Y 399.335,Z 496.715,A -85,B 0,C 180,E1 -11265.048,E2 -11265.048} C_VEL
LIN {X 0,Y 400.135,Z 486.159,A -85,B 0,C 180,E1 -11265.931,E2 -11265.931} C_VEL
LIN {X 0,Y 400.959,Z 473.462,A -85,B 0,C 180,E1 -11266.747,E2 -11266.747} C_VEL
LIN {X 0,Y 401.688,Z 460.815,A -85,B 0,C 180,E1 -11267.339,E2 -11267.339} C_VEL
LIN {X 0,Y 402.092,Z 448.877,A -85,B 0,C 180,E1 -11267.714,E2 -11267.714} C_VEL
LIN {X 0,Y 403.234,Z 370.363,A -85,B 0,C 180,E1 -11269.169,E2 -11269.169} C_VEL
LIN {X 0,Y 398.837,Z 341.203,A -85,B 0,C 180,E1 -11269.952,E2 -11269.952} C_VEL
LIN {X 0,Y 400.125,Z 323.608,A -85,B 0,C 180,E1 -11273.555,E2 -11273.555} C_VEL
LIN {X 0,Y 400.505,Z 318.254,A -85,B 0,C 180,E1 -11274.664,E2 -11274.664} C_VEL
LIN {X 0,Y 398.646,Z 307.833,A -85,B 0,C 180,E1 -11277,E2 -11277} C_VEL
LIN {X 0,Y 397.176,Z 301.013,A -85,B 0,C 180,E1 -11278.613,E2 -11278.613} C_VEL
LIN {X 0,Y 397.084,Z 301.025,A -85,B 0,C 180,E1 -11282.072,E2 -11282.072} C_VEL
LIN {X 0,Y 397.124,Z 301.014,A -85,B 0,C 180,E1 -11285.504,E2 -11285.504} C_VEL
LIN {X 0,Y 397.129,Z 301.014,A -85,B 0,C 180,E1 -11288.861,E2 -11288.861} C_VEL
LIN {X 0,Y 397.071,Z 301.026,A -85,B 0,C 180,E1 -11292.268,E2 -11292.268} C_VEL
LIN {X 0,Y 397.089,Z 301.018,A -85,B 0,C 180,E1 -11295.069,E2 -11295.069} C_VEL
LIN {X 0,Y 397.067,Z 301.022,A -85,B 0,C 180,E1 -11298.022,E2 -11298.022} C_VEL
LIN {X 0,Y 397.131,Z 301.013,A -85,B 0,C 180,E1 -11301.139,E2 -11301.139} C_VEL
LIN {X 0,Y 397.119,Z 301.019,A -85,B 0,C 180,E1 -11304.497,E2 -11304.497} C_VEL
LIN {X 0,Y 397.077,Z 301.019,A -85,B 0,C 180,E1 -11307.928,E2 -11307.928} C_VEL
LIN {X 0,Y 397.12,Z 301.014,A -85,B 0,C 180,E1 -11311.456,E2 -11311.456} C_VEL
LIN {X 0,Y 397.151,Z 301.013,A -85,B 0,C 180,E1 -11314.488,E2 -11314.488} C_VEL
LIN {X 0,Y 397.106,Z 301.021,A -85,B 0,C 180,E1 -11317.085,E2 -11317.085} C_VEL
LIN {X 0,Y 397.144,Z 301.011,A -85,B 0,C 180,E1 -11320.353,E2 -11320.353} C_VEL
LIN {X 0,Y 397.162,Z 301.011,A -85,B 0,C 180,E1 -11323.553,E2 -11323.553} C_VEL
LIN {X 0,Y 397.226,Z 301.003,A -85,B 0,C 180,E1 -11326.703,E2 -11326.703} C_VEL
LIN {X 0,Y 397.211,Z 301.004,A -85,B 0,C 180,E1 -11329.809,E2 -11329.809} C_VEL
LIN {X 0,Y 397.348,Z 300.988,A -85,B 0,C 180,E1 -11332.888,E2 -11332.888} C_VEL
LIN {X 0,Y 397.243,Z 301.001,A -85,B 0,C 180,E1 -11334.925,E2 -11334.925} C_VEL
LIN {X 0,Y 397.44,Z 300.975,A -85,B 0,C 180,E1 -11337.973,E2 -11337.973} C_VEL
LIN {X 0,Y 397.568,Z 300.96,A -85,B 0,C 180,E1 -11340,E2 -11340} C_VEL
LIN {X 0,Y 397.365,Z 300.985,A -85,B 0,C 180,E1 -11343.042,E2 -11343.042} C_VEL
LIN {X 0,Y 397.295,Z 300.992,A -85,B 0,C 180,E1 -11346.515,E2 -11346.515} C_VEL
LIN {X 0,Y 397.229,Z 301.001,A -85,B 0,C 180,E1 -11349.162,E2 -11349.162} C_VEL
LIN {X 0,Y 397.213,Z 301.004,A -85,B 0,C 180,E1 -11352.258,E2 -11352.258} C_VEL
LIN {X 0,Y 397.171,Z 301.009,A -85,B 0,C 180,E1 -11355.392,E2 -11355.392} C_VEL
LIN {X 0,Y 397.152,Z 301.01,A -85,B 0,C 180,E1 -11358.574,E2 -11358.574} C_VEL
LIN {X 0,Y 397.09,Z 301.022,A -85,B 0,C 180,E1 -11361.819,E2 -11361.819} C_VEL
LIN {X 0,Y 397.099,Z 301.016,A -85,B 0,C 180,E1 -11365.136,E2 -11365.136} C_VEL
LIN {X 0,Y 397.06,Z 301.024,A -85,B 0,C 180,E1 -11368.549,E2 -11368.549} C_VEL
LIN {X 0,Y 397.077,Z 301.022,A -85,B 0,C 180,E1 -11371.835,E2 -11371.835} C_VEL
LIN {X 0,Y 397.115,Z 301.019,A -85,B 0,C 180,E1 -11374.495,E2 -11374.495} C_VEL
LIN {X 0,Y 397.085,Z 301.024,A -85,B 0,C 180,E1 -11378.277,E2 -11378.277} C_VEL
LIN {X 0,Y 397.048,Z 301.024,A -85,B 0,C 180,E1 -11381.975,E2 -11381.975} C_VEL
LIN {X 0,Y 397.076,Z 301.021,A -85,B 0,C 180,E1 -11385.071,E2 -11385.071} C_VEL
LIN {X 0,Y 397.047,Z 301.025,A -85,B 0,C 180,E1 -11389.085,E2 -11389.085} C_VEL
LIN {X 0,Y 397.083,Z 301.018,A -85,B 0,C 180,E1 -11391.722,E2 -11391.722} C_VEL
LIN {X 0,Y 397.032,Z 301.029,A -85,B 0,C 180,E1 -11394.515,E2 -11394.515} C_VEL
LIN {X 0,Y 397.068,Z 301.02,A -85,B 0,C 180,E1 -11397.926,E2 -11397.926} C_VEL
LIN {X 0,Y 397.117,Z 301.015,A -85,B 0,C 180,E1 -11400.294,E2 -11400.294} C_VEL
LIN {X 0,Y 397.073,Z 301.02,A -85,B 0,C 180,E1 -11403.736,E2 -11403.736} C_VEL
LIN {X 0,Y 397.105,Z 301.023,A -85,B 0,C 180,E1 -11407.084,E2 -11407.084} C_VEL
LIN {X 0,Y 397.152,Z 301.01,A -85,B 0,C 180,E1 -11410.351,E2 -11410.351} C_VEL
LIN {X 0,Y 397.17,Z 301.011,A -85,B 0,C 180,E1 -11413.551,E2 -11413.551} C_VEL
LIN {X 0,Y 397.235,Z 301,A -85,B 0,C 180,E1 -11416.7,E2 -11416.7} C_VEL
LIN {X 0,Y 397.214,Z 301.004,A -85,B 0,C 180,E1 -11419.806,E2 -11419.806} C_VEL
LIN {X 0,Y 397.297,Z 300.993,A -85,B 0,C 180,E1 -11422.884,E2 -11422.884} C_VEL
LIN {X 0,Y 397.232,Z 301.001,A -85,B 0,C 180,E1 -11424.922,E2 -11424.922} C_VEL
LIN {X 0,Y 397.442,Z 300.976,A -85,B 0,C 180,E1 -11427.97,E2 -11427.97} C_VEL
LIN {X 0,Y 397.32,Z 300.99,A -85,B 0,C 180,E1 -11431.01,E2 -11431.01} C_VEL
LIN {X 0,Y 397.326,Z 300.989,A -85,B 0,C 180,E1 -11433.038,E2 -11433.038} C_VEL
LIN {X 0,Y 397.327,Z 300.995,A -85,B 0,C 180,E1 -11436.088,E2 -11436.088} C_VEL
LIN {X 0,Y 397.255,Z 301.115,A -85,B 0,C 180,E1 -11439.062,E2 -11439.062} C_VEL
LIN {X 0,Y 399.166,Z 311.461,A -85,B 0,C 180,E1 -11441.678,E2 -11441.678} C_VEL
LIN {X 0,Y 399.205,Z 313.334,A -85,B 0,C 180,E1 -11442.128,E2 -11442.128} C_VEL
LIN {X 0,Y 403.577,Z 335.508,A -85,B 0,C 180,E1 -11442.786,E2 -11442.786} C_VEL
LIN {X 0,Y 402.524,Z 404.4,A -85,B 0,C 180,E1 -11444.046,E2 -11444.046} C_VEL
LIN {X 0,Y 401.77,Z 408.324,A -85,B 0,C 180,E1 -11444.086,E2 -11444.086} C_VEL
LIN {X 0,Y 395.976,Z 420.56,A -85,B 0,C 180,E1 -11444.093,E2 -11444.093} C_VEL
LIN {X 0,Y 395.352,Z 424.434,A -85,B 0,C 180,E1 -11444.18,E2 -11444.18} C_VEL
LIN {X 0,Y 394.871,Z 437.662,A -85,B 0,C 180,E1 -11444.688,E2 -11444.688} C_VEL
LIN {X 0,Y 394.32,Z 449.868,A -85,B 0,C 180,E1 -11445.369,E2 -11445.369} C_VEL
LIN {X 0,Y 393.609,Z 460.684,A -85,B 0,C 180,E1 -11446.157,E2 -11446.157} C_VEL
LIN {X 0,Y 392.844,Z 471.614,A -85,B 0,C 180,E1 -11447.164,E2 -11447.164} C_VEL
LIN {X 0,Y 392.04,Z 480.519,A -85,B 0,C 180,E1 -11448.172,E2 -11448.172} C_VEL
LIN {X 0,Y 391.359,Z 489.417,A -85,B 0,C 180,E1 -11449.399,E2 -11449.399} C_VEL
LIN {X 0,Y 390.698,Z 497.231,A -85,B 0,C 180,E1 -11450.708,E2 -11450.708} C_VEL
LIN {X 0,Y 390.048,Z 504.635,A -85,B 0,C 180,E1 -11452.228,E2 -11452.228} C_VEL
LIN {X 0,Y 389.556,Z 511.278,A -85,B 0,C 180,E1 -11453.944,E2 -11453.944} C_VEL
LIN {X 0,Y 389.182,Z 516.464,A -85,B 0,C 180,E1 -11455.678,E2 -11455.678} C_VEL
LIN {X 0,Y 388.81,Z 520.693,A -85,B 0,C 180,E1 -11457.661,E2 -11457.661} C_VEL
LIN {X 0,Y 388.613,Z 523.484,A -85,B 0,C 180,E1 -11459.764,E2 -11459.764} C_VEL
LIN {X 0,Y 388.535,Z 524.545,A -85,B 0,C 180,E1 -11461.771,E2 -11461.771} C_VEL
LIN {X 0,Y 388.557,Z 524.197,A -85,B 0,C 180,E1 -11463.693,E2 -11463.693} C_VEL
LIN {X 0,Y 388.722,Z 522.548,A -85,B 0,C 180,E1 -11465.551,E2 -11465.551} C_VEL
LIN {X 0,Y 389.004,Z 519.656,A -85,B 0,C 180,E1 -11467.351,E2 -11467.351} C_VEL
LIN {X 0,Y 389.333,Z 515.371,A -85,B 0,C 180,E1 -11469.175,E2 -11469.175} C_VEL
LIN {X 0,Y 389.758,Z 510.376,A -85,B 0,C 180,E1 -11470.77,E2 -11470.77} C_VEL
LIN {X 0,Y 390.412,Z 503.74,A -85,B 0,C 180,E1 -11472.433,E2 -11472.433} C_VEL
LIN {X 0,Y 391.189,Z 495.484,A -85,B 0,C 180,E1 -11474.058,E2 -11474.058} C_VEL
LIN {X 0,Y 392.023,Z 487.135,A -85,B 0,C 180,E1 -11475.387,E2 -11475.387} C_VEL
LIN {X 0,Y 392.904,Z 477.833,A -85,B 0,C 180,E1 -11476.599,E2 -11476.599} C_VEL
LIN {X 0,Y 393.655,Z 468.163,A -85,B 0,C 180,E1 -11477.632,E2 -11477.632} C_VEL
LIN {X 0,Y 394.526,Z 457.222,A -85,B 0,C 180,E1 -11478.562,E2 -11478.562} C_VEL
LIN {X 0,Y 395.293,Z 444.946,A -85,B 0,C 180,E1 -11479.369,E2 -11479.369} C_VEL
LIN {X 0,Y 395.902,Z 432.208,A -85,B 0,C 180,E1 -11479.982,E2 -11479.982} C_VEL
LIN {X 0,Y 396.296,Z 419.723,A -85,B 0,C 180,E1 -11480.373,E2 -11480.373} C_VEL
LIN {X 0,Y 397.606,Z 335.44,A -85,B 0,C 180,E1 -11481.987,E2 -11481.987} C_VEL
LIN {X 0,Y 393.16,Z 315.509,A -85,B 0,C 180,E1 -11482.652,E2 -11482.652} C_VEL
LIN {X 0,Y 392.5,Z 313.534,A -85,B 0,C 180,E1 -11482.739,E2 -11482.739} C_VEL
LIN {X 0,Y 390.072,Z 301.898,A -85,B 0,C 180,E1 -11485.508,E2 -11485.508} C_VEL
LIN {X 0,Y 389.987,Z 301.908,A -85,B 0,C 180,E1 -11488.492,E2 -11488.492} C_VEL
LIN {X 0,Y 390.077,Z 301.9,A -85,B 0,C 180,E1 -11492.067,E2 -11492.067} C_VEL
LIN {X 0,Y 390.036,Z 301.905,A -85,B 0,C 180,E1 -11495.516,E2 -11495.516} C_VEL
LIN {X 0,Y 390.01,Z 301.907,A -85,B 0,C 180,E1 -11498.875,E2 -11498.875} C_VEL
LIN {X 0,Y 390.081,Z 301.896,A -85,B 0,C 180,E1 -11502.164,E2 -11502.164} C_VEL
LIN {X 0,Y 390.095,Z 301.892,A -85,B 0,C 180,E1 -11505.391,E2 -11505.391} C_VEL
LIN {X 0,Y 390.099,Z 301.894,A -85,B 0,C 180,E1 -11508.57,E2 -11508.57} C_VEL
LIN {X 0,Y 390.259,Z 301.87,A -85,B 0,C 180,E1 -11512.031,E2 -11512.031} C_VEL
LIN {X 0,Y 390.175,Z 301.883,A -85,B 0,C 180,E1 -11514.833,E2 -11514.833} C_VEL
LIN {X 0,Y 390.371,Z 301.855,A -85,B 0,C 180,E1 -11517.936,E2 -11517.936} C_VEL
LIN {X 0,Y 390.499,Z 301.833,A -85,B 0,C 180,E1 -11520,E2 -11520} C_VEL
LIN {X 0,Y 390.272,Z 301.866,A -85,B 0,C 180,E1 -11523.097,E2 -11523.097} C_VEL
LIN {X 0,Y 390.279,Z 301.867,A -85,B 0,C 180,E1 -11526.203,E2 -11526.203} C_VEL
LIN {X 0,Y 390.162,Z 301.886,A -85,B 0,C 180,E1 -11529.33,E2 -11529.33} C_VEL
LIN {X 0,Y 390.131,Z 301.879,A -85,B 0,C 180,E1 -11532.484,E2 -11532.484} C_VEL
LIN {X 0,Y 390.097,Z 301.885,A -85,B 0,C 180,E1 -11535.679,E2 -11535.679} C_VEL
LIN {X 0,Y 390.073,Z 301.895,A -85,B 0,C 180,E1 -11538.924,E2 -11538.924} C_VEL
LIN {X 0,Y 390.06,Z 301.892,A -85,B 0,C 180,E1 -11542.233,E2 -11542.233} C_VEL
LIN {X 0,Y 390.077,Z 301.893,A -85,B 0,C 180,E1 -11545.746,E2 -11545.746} C_VEL
LIN {X 0,Y 390.023,Z 301.896,A -85,B 0,C 180,E1 -11549.113,E2 -11549.113} C_VEL
LIN {X 0,Y 390.005,Z 301.9,A -85,B 0,C 180,E1 -11552.725,E2 -11552.725} C_VEL
LIN {X 0,Y 390.024,Z 301.902,A -85,B 0,C 180,E1 -11555.83,E2 -11555.83} C_VEL
LIN {X 0,Y 390.067,Z 301.895,A -85,B 0,C 180,E1 -11559.228,E2 -11559.228} C_VEL
LIN {X 0,Y 390.091,Z 301.895,A -85,B 0,C 180,E1 -11562.391,E2 -11562.391} C_VEL
LIN {X 0,Y 390.089,Z 301.899,A -85,B 0,C 180,E1 -11565.37,E2 -11565.37} C_VEL
LIN {X 0,Y 390.078,Z 301.897,A -85,B 0,C 180,E1 -11568.201,E2 -11568.201} C_VEL
LIN {X 0,Y 390.072,Z 301.896,A -85,B 0,C 180,E1 -11570.913,E2 -11570.913} C_VEL
LIN {X 0,Y 390.065,Z 301.898,A -85,B 0,C 180,E1 -11574.798,E2 -11574.798} C_VEL
LIN {X 0,Y 390.009,Z 301.908,A -85,B 0,C 180,E1 -11578.501,E2 -11578.501} C_VEL
LIN {X 0,Y 390.145,Z 302.081,A -85,B 0,C 180,E1 -11581.164,E2 -11581.164} C_VEL
LIN {X 0,Y 392.864,Z 314.599,A -85,B 0,C 180,E1 -11584.054,E2 -11584.054} C_VEL
LIN {X 0,Y 393.665,Z 319.776,A -85,B 0,C 180,E1 -11585.201,E2 -11585.201} C_VEL
LIN {X 0,Y 392.475,Z 335.371,A -85,B 0,C 180,E1 -11588.376,E2 -11588.376} C_VEL
LIN {X 0,Y 392.173,Z 339.828,A -85,B 0,C 180,E1 -11589.277,E2 -11589.277} C_VEL
LIN {X 0,Y 396.087,Z 363.134,A -85,B 0,C 180,E1 -11589.989,E2 -11589.989} C_VEL
LIN {X 0,Y 397.229,Z 371.654,A -85,B 0,C 180,E1 -11590.223,E2 -11590.223} C_VEL
LIN {X 0,Y 395.928,Z 449.136,A -85,B 0,C 180,E1 -11591.706,E2 -11591.706} C_VEL
LIN {X 0,Y 395.281,Z 462.902,A -85,B 0,C 180,E1 -11592.178,E2 -11592.178} C_VEL
LIN {X 0,Y 394.469,Z 475.854,A -85,B 0,C 180,E1 -11592.842,E2 -11592.842} C_VEL
LIN {X 0,Y 393.562,Z 487.652,A -85,B 0,C 180,E1 -11593.67,E2 -11593.67} C_VEL
LIN {X 0,Y 392.672,Z 499.047,A -85,B 0,C 180,E1 -11594.697,E2 -11594.697} C_VEL
LIN {X 0,Y 391.736,Z 509.807,A -85,B 0,C 180,E1 -11595.917,E2 -11595.917} C_VEL
LIN {X 0,Y 390.858,Z 519.431,A -85,B 0,C 180,E1 -11597.28,E2 -11597.28} C_VEL
LIN {X 0,Y 389.978,Z 528.324,A -85,B 0,C 180,E1 -11598.834,E2 -11598.834} C_VEL
LIN {X 0,Y 389.446,Z 535.455,A -85,B 0,C 180,E1 -11600.395,E2 -11600.395} C_VEL
LIN {X 0,Y 389.014,Z 541.982,A -85,B 0,C 180,E1 -11602.217,E2 -11602.217} C_VEL
LIN {X 0,Y 388.772,Z 546.494,A -85,B 0,C 180,E1 -11603.859,E2 -11603.859} C_VEL
LIN {X 0,Y 388.739,Z 548.589,A -85,B 0,C 180,E1 -11604.817,E2 -11604.817} C_VEL
LIN {X 0,Y 388.7,Z 550.412,A -85,B 0,C 180,E1 -11605.856,E2 -11605.856} C_VEL
LIN {X 0,Y 388.701,Z 552.78,A -85,B 0,C 180,E1 -11607.931,E2 -11607.931} C_VEL
LIN {X 0,Y 388.739,Z 553.372,A -85,B 0,C 180,E1 -11608.968,E2 -11608.968} C_VEL
LIN {X 0,Y 388.727,Z 553.529,A -85,B 0,C 180,E1 -11610.003,E2 -11610.003} C_VEL
LIN {X 0,Y 388.74,Z 553.276,A -85,B 0,C 180,E1 -11611.039,E2 -11611.039} C_VEL
LIN {X 0,Y 388.703,Z 552.63,A -85,B 0,C 180,E1 -11612.076,E2 -11612.076} C_VEL
LIN {X 0,Y 388.642,Z 551.588,A -85,B 0,C 180,E1 -11613.113,E2 -11613.113} C_VEL
LIN {X 0,Y 388.702,Z 550.097,A -85,B 0,C 180,E1 -11614.15,E2 -11614.15} C_VEL
LIN {X 0,Y 388.728,Z 546.937,A -85,B 0,C 180,E1 -11615.755,E2 -11615.755} C_VEL
LIN {X 0,Y 388.935,Z 542.931,A -85,B 0,C 180,E1 -11617.27,E2 -11617.27} C_VEL
LIN {X 0,Y 389.257,Z 536.607,A -85,B 0,C 180,E1 -11619.092,E2 -11619.092} C_VEL
LIN {X 0,Y 389.727,Z 529.716,A -85,B 0,C 180,E1 -11620.654,E2 -11620.654} C_VEL
LIN {X 0,Y 390.478,Z 521.11,A -85,B 0,C 180,E1 -11622.212,E2 -11622.212} C_VEL
LIN {X 0,Y 391.204,Z 512.255,A -85,B 0,C 180,E1 -11623.508,E2 -11623.508} C_VEL
LIN {X 0,Y 392.076,Z 501.357,A -85,B 0,C 180,E1 -11624.802,E2 -11624.802} C_VEL
LIN {X 0,Y 392.906,Z 490.397,A -85,B 0,C 180,E1 -11625.832,E2 -11625.832} C_VEL
LIN {X 0,Y 393.787,Z 478.12,A -85,B 0,C 180,E1 -11626.728,E2 -11626.728} C_VEL
LIN {X 0,Y 394.581,Z 465.237,A -85,B 0,C 180,E1 -11627.427,E2 -11627.427} C_VEL
LIN {X 0,Y 395.173,Z 452.28,A -85,B 0,C 180,E1 -11627.901,E2 -11627.901} C_VEL
LIN {X 0,Y 395.588,Z 432.552,A -85,B 0,C 180,E1 -11628.317,E2 -11628.317} C_VEL
LIN {X 0,Y 396.321,Z 369.97,A -85,B 0,C 180,E1 -11629.493,E2 -11629.493} C_VEL
LIN {X 0,Y 391.946,Z 340.933,A -85,B 0,C 180,E1 -11630.297,E2 -11630.297} C_VEL
LIN {X 0,Y 393.319,Z 323.243,A -85,B 0,C 180,E1 -11633.988,E2 -11633.988} C_VEL
LIN {X 0,Y 393.539,Z 319.336,A -85,B 0,C 180,E1 -11634.815,E2 -11634.815} C_VEL
LIN {X 0,Y 391.621,Z 308.754,A -85,B 0,C 180,E1 -11637.235,E2 -11637.235} C_VEL
LIN {X 0,Y 390.144,Z 301.889,A -85,B 0,C 180,E1 -11638.91,E2 -11638.91} C_VEL
LIN {X 0,Y 390.048,Z 301.896,A -85,B 0,C 180,E1 -11642.722,E2 -11642.722} C_VEL
LIN {X 0,Y 390.06,Z 301.896,A -85,B 0,C 180,E1 -11645.826,E2 -11645.826} C_VEL
LIN {X 0,Y 390.07,Z 301.892,A -85,B 0,C 180,E1 -11649.218,E2 -11649.218} C_VEL
LIN {X 0,Y 390.045,Z 301.902,A -85,B 0,C 180,E1 -11652.374,E2 -11652.374} C_VEL
LIN {X 0,Y 390.046,Z 301.895,A -85,B 0,C 180,E1 -11655.354,E2 -11655.354} C_VEL
LIN {X 0,Y 390.032,Z 301.9,A -85,B 0,C 180,E1 -11658.187,E2 -11658.187} C_VEL
LIN {X 0,Y 390.091,Z 301.892,A -85,B 0,C 180,E1 -11660.908,E2 -11660.908} C_VEL
LIN {X 0,Y 390.085,Z 301.896,A -85,B 0,C 180,E1 -11664.793,E2 -11664.793} C_VEL
LIN {X 0,Y 390.023,Z 301.902,A -85,B 0,C 180,E1 -11668.495,E2 -11668.495} C_VEL
LIN {X 0,Y 390.117,Z 301.886,A -85,B 0,C 180,E1 -11672.07,E2 -11672.07} C_VEL
LIN {X 0,Y 390.077,Z 301.892,A -85,B 0,C 180,E1 -11675.519,E2 -11675.519} C_VEL
LIN {X 0,Y 390.052,Z 301.9,A -85,B 0,C 180,E1 -11678.878,E2 -11678.878} C_VEL
LIN {X 0,Y 390.109,Z 301.887,A -85,B 0,C 180,E1 -11682.166,E2 -11682.166} C_VEL
LIN {X 0,Y 390.138,Z 301.888,A -85,B 0,C 180,E1 -11685.392,E2 -11685.392} C_VEL
LIN {X 0,Y 390.141,Z 301.884,A -85,B 0,C 180,E1 -11688.571,E2 -11688.571} C_VEL
LIN {X 0,Y 390.304,Z 301.863,A -85,B 0,C 180,E1 -11692.032,E2 -11692.032} C_VEL
LIN {X 0,Y 390.216,Z 301.875,A -85,B 0,C 180,E1 -11694.833,E2 -11694.833} C_VEL
LIN {X 0,Y 390.409,Z 301.851,A -85,B 0,C 180,E1 -11697.937,E2 -11697.937} C_VEL
LIN {X 0,Y 390.538,Z 301.835,A -85,B 0,C 180,E1 -11700,E2 -11700} C_VEL
LIN {X 0,Y 390.3,Z 301.865,A -85,B 0,C 180,E1 -11703.097,E2 -11703.097} C_VEL
LIN {X 0,Y 390.255,Z 301.869,A -85,B 0,C 180,E1 -11706.506,E2 -11706.506} C_VEL
LIN {X 0,Y 390.187,Z 301.88,A -85,B 0,C 180,E1 -11709.329,E2 -11709.329} C_VEL
LIN {X 0,Y 390.165,Z 301.881,A -85,B 0,C 180,E1 -11712.483,E2 -11712.483} C_VEL
LIN {X 0,Y 390.133,Z 301.889,A -85,B 0,C 180,E1 -11715.677,E2 -11715.677} C_VEL
LIN {X 0,Y 390.097,Z 301.888,A -85,B 0,C 180,E1 -11718.923,E2 -11718.923} C_VEL
LIN {X 0,Y 390.031,Z 301.901,A -85,B 0,C 180,E1 -11722.235,E2 -11722.235} C_VEL
LIN {X 0,Y 390.049,Z 301.897,A -85,B 0,C 180,E1 -11725.722,E2 -11725.722} C_VEL
LIN {X 0,Y 390.021,Z 301.898,A -85,B 0,C 180,E1 -11729.113,E2 -11729.113} C_VEL
LIN {X 0,Y 390.039,Z 301.898,A -85,B 0,C 180,E1 -11732.722,E2 -11732.722} C_VEL
LIN {X 0,Y 390.04,Z 301.897,A -85,B 0,C 180,E1 -11735.822,E2 -11735.822} C_VEL
LIN {X 0,Y 390.028,Z 301.897,A -85,B 0,C 180,E1 -11739.21,E2 -11739.21} C_VEL
LIN {X 0,Y 390.028,Z 301.903,A -85,B 0,C 180,E1 -11742.371,E2 -11742.371} C_VEL
LIN {X 0,Y 390.008,Z 301.9,A -85,B 0,C 180,E1 -11745.348,E2 -11745.348} C_VEL
LIN {X 0,Y 390.006,Z 301.902,A -85,B 0,C 180,E1 -11748.182,E2 -11748.182} C_VEL
LIN {X 0,Y 390.051,Z 301.899,A -85,B 0,C 180,E1 -11750.902,E2 -11750.902} C_VEL
LIN {X 0,Y 389.988,Z 301.903,A -85,B 0,C 180,E1 -11754.189,E2 -11754.189} C_VEL
LIN {X 0,Y 390.018,Z 301.901,A -85,B 0,C 180,E1 -11757.275,E2 -11757.275} C_VEL
LIN {X 0,Y 390.026,Z 301.904,A -85,B 0,C 180,E1 -11760.886,E2 -11760.886} C_VEL
LIN {X 0,Y 390.066,Z 301.893,A -85,B 0,C 180,E1 -11764.377,E2 -11764.377} C_VEL
LIN {X 0,Y 390.04,Z 301.896,A -85,B 0,C 180,E1 -11767.764,E2 -11767.764} C_VEL
LIN {X 0,Y 390.108,Z 301.893,A -85,B 0,C 180,E1 -11771.076,E2 -11771.076} C_VEL
LIN {X 0,Y 390.14,Z 301.883,A -85,B 0,C 180,E1 -11774.321,E2 -11774.321} C_VEL
LIN {X 0,Y 390.175,Z 301.884,A -85,B 0,C 180,E1 -11777.515,E2 -11777.515} C_VEL
LIN {X 0,Y 390.192,Z 301.877,A -85,B 0,C 180,E1 -11780.668,E2 -11780.668} C_VEL
LIN {X 0,Y 390.28,Z 301.869,A -85,B 0,C 180,E1 -11783.794,E2 -11783.794} C_VEL
LIN {X 0,Y 390.409,Z 301.853,A -85,B 0,C 180,E1 -11787.934,E2 -11787.934} C_VEL
LIN {X 0,Y 390.291,Z 301.865,A -85,B 0,C 180,E1 -11791.028,E2 -11791.028} C_VEL
LIN {X 0,Y 390.263,Z 301.869,A -85,B 0,C 180,E1 -11793.093,E2 -11793.093} C_VEL
LIN {X 0,Y 390.28,Z 301.872,A -85,B 0,C 180,E1 -11796.199,E2 -11796.199} C_VEL
LIN {X 0,Y 390.219,Z 301.936,A -85,B 0,C 180,E1 -11798.802,E2 -11798.802} C_VEL
LIN {X 0,Y 392.217,Z 313.017,A -85,B 0,C 180,E1 -11801.652,E2 -11801.652} C_VEL
LIN {X 0,Y 392.264,Z 313.808,A -85,B 0,C 180,E1 -11801.812,E2 -11801.812} C_VEL
LIN {X 0,Y 396.824,Z 336.242,A -85,B 0,C 180,E1 -11802.481,E2 -11802.481} C_VEL
LIN {X 0,Y 395.457,Z 420.697,A -85,B 0,C 180,E1 -11804.074,E2 -11804.074} C_VEL
LIN {X 0,Y 395.352,Z 424.434,A -85,B 0,C 180,E1 -11804.18,E2 -11804.18} C_VEL
LIN {X 0,Y 394.699,Z 428.306,A -85,B 0,C 180,E1 -11804.277,E2 -11804.277} C_VEL
LIN {X 0,Y 391.722,Z 434.343,A -85,B 0,C 180,E1 -11804.385,E2 -11804.385} C_VEL
LIN {X 0,Y 388.617,Z 440.277,A -85,B 0,C 180,E1 -11804.544,E2 -11804.544} C_VEL
LIN {X 0,Y 387.769,Z 443.992,A -85,B 0,C 180,E1 -11804.72,E2 -11804.72} C_VEL
LIN {X 0,Y 387.142,Z 456.234,A -85,B 0,C 180,E1 -11805.527,E2 -11805.527} C_VEL
LIN {X 0,Y 386.193,Z 467.878,A -85,B 0,C 180,E1 -11806.515,E2 -11806.515} C_VEL
LIN {X 0,Y 385.352,Z 478.3,A -85,B 0,C 180,E1 -11807.645,E2 -11807.645} C_VEL
LIN {X 0,Y 384.56,Z 488.017,A -85,B 0,C 180,E1 -11808.949,E2 -11808.949} C_VEL
LIN {X 0,Y 383.761,Z 496.579,A -85,B 0,C 180,E1 -11810.357,E2 -11810.357} C_VEL
LIN {X 0,Y 383.149,Z 503.715,A -85,B 0,C 180,E1 -11811.799,E2 -11811.799} C_VEL
LIN {X 0,Y 382.662,Z 509.815,A -85,B 0,C 180,E1 -11813.32,E2 -11813.32} C_VEL
LIN {X 0,Y 382.239,Z 515.175,A -85,B 0,C 180,E1 -11815.011,E2 -11815.011} C_VEL
LIN {X 0,Y 381.889,Z 519.443,A -85,B 0,C 180,E1 -11816.794,E2 -11816.794} C_VEL
LIN {X 0,Y 381.594,Z 522.47,A -85,B 0,C 180,E1 -11818.605,E2 -11818.605} C_VEL
LIN {X 0,Y 381.501,Z 523.961,A -85,B 0,C 180,E1 -11820.022,E2 -11820.022} C_VEL
LIN {X 0,Y 381.434,Z 524.856,A -85,B 0,C 180,E1 -11822.052,E2 -11822.052} C_VEL
LIN {X 0,Y 381.476,Z 524.324,A -85,B 0,C 180,E1 -11823.999,E2 -11823.999} C_VEL
LIN {X 0,Y 381.676,Z 522.485,A -85,B 0,C 180,E1 -11825.885,E2 -11825.885} C_VEL
LIN {X 0,Y 381.982,Z 519.458,A -85,B 0,C 180,E1 -11827.707,E2 -11827.707} C_VEL
LIN {X 0,Y 382.321,Z 515.295,A -85,B 0,C 180,E1 -11829.46,E2 -11829.46} C_VEL
LIN {X 0,Y 382.902,Z 509.231,A -85,B 0,C 180,E1 -11831.35,E2 -11831.35} C_VEL
LIN {X 0,Y 383.635,Z 501.943,A -85,B 0,C 180,E1 -11833.094,E2 -11833.094} C_VEL
LIN {X 0,Y 384.548,Z 493.789,A -85,B 0,C 180,E1 -11834.645,E2 -11834.645} C_VEL
LIN {X 0,Y 385.379,Z 485.218,A -85,B 0,C 180,E1 -11835.965,E2 -11835.965} C_VEL
LIN {X 0,Y 386.314,Z 474.881,A -85,B 0,C 180,E1 -11837.257,E2 -11837.257} C_VEL
LIN {X 0,Y 387.242,Z 464.825,A -85,B 0,C 180,E1 -11838.267,E2 -11838.267} C_VEL
LIN {X 0,Y 388.085,Z 452.825,A -85,B 0,C 180,E1 -11839.227,E2 -11839.227} C_VEL
LIN {X 0,Y 388.854,Z 440.216,A -85,B 0,C 180,E1 -11839.975,E2 -11839.975} C_VEL
LIN {X 0,Y 389.426,Z 426.926,A -85,B 0,C 180,E1 -11840.531,E2 -11840.531} C_VEL
LIN {X 0,Y 389.801,Z 412.322,A -85,B 0,C 180,E1 -11840.886,E2 -11840.886} C_VEL
LIN {X 0,Y 391.095,Z 336.9,A -85,B 0,C 180,E1 -11842.339,E2 -11842.339} C_VEL
LIN {X 0,Y 386.992,Z 318.23,A -85,B 0,C 180,E1 -11842.977,E2 -11842.977} C_VEL
LIN {X 0,Y 385.348,Z 313.751,A -85,B 0,C 180,E1 -11843.199,E2 -11843.199} C_VEL
LIN {X 0,Y 383.01,Z 302.779,A -85,B 0,C 180,E1 -11845.874,E2 -11845.874} C_VEL
LIN {X 0,Y 382.962,Z 302.783,A -85,B 0,C 180,E1 -11849.588,E2 -11849.588} C_VEL
LIN {X 0,Y 383.016,Z 302.78,A -85,B 0,C 180,E1 -11852.695,E2 -11852.695} C_VEL
LIN {X 0,Y 383.009,Z 302.781,A -85,B 0,C 180,E1 -11855.037,E2 -11855.037} C_VEL
LIN {X 0,Y 382.947,Z 302.788,A -85,B 0,C 180,E1 -11858.466,E2 -11858.466} C_VEL
LIN {X 0,Y 383.016,Z 302.774,A -85,B 0,C 180,E1 -11861.824,E2 -11861.824} C_VEL
LIN {X 0,Y 383.061,Z 302.769,A -85,B 0,C 180,E1 -11865.116,E2 -11865.116} C_VEL
LIN {X 0,Y 383.048,Z 302.772,A -85,B 0,C 180,E1 -11868.356,E2 -11868.356} C_VEL
LIN {X 0,Y 383.216,Z 302.747,A -85,B 0,C 180,E1 -11871.975,E2 -11871.975} C_VEL
LIN {X 0,Y 383.147,Z 302.76,A -85,B 0,C 180,E1 -11874.738,E2 -11874.738} C_VEL
LIN {X 0,Y 383.338,Z 302.731,A -85,B 0,C 180,E1 -11877.899,E2 -11877.899} C_VEL
LIN {X 0,Y 383.469,Z 302.708,A -85,B 0,C 180,E1 -11880,E2 -11880} C_VEL
LIN {X 0,Y 383.208,Z 302.745,A -85,B 0,C 180,E1 -11883.154,E2 -11883.154} C_VEL
LIN {X 0,Y 383.235,Z 302.745,A -85,B 0,C 180,E1 -11886.317,E2 -11886.317} C_VEL
LIN {X 0,Y 383.109,Z 302.763,A -85,B 0,C 180,E1 -11889.503,E2 -11889.503} C_VEL
LIN {X 0,Y 383.095,Z 302.757,A -85,B 0,C 180,E1 -11892.718,E2 -11892.718} C_VEL
LIN {X 0,Y 383.038,Z 302.763,A -85,B 0,C 180,E1 -11895.975,E2 -11895.975} C_VEL
LIN {X 0,Y 383.031,Z 302.769,A -85,B 0,C 180,E1 -11899.285,E2 -11899.285} C_VEL
LIN {X 0,Y 383.007,Z 302.772,A -85,B 0,C 180,E1 -11902.665,E2 -11902.665} C_VEL
LIN {X 0,Y 383.038,Z 302.768,A -85,B 0,C 180,E1 -11906.126,E2 -11906.126} C_VEL
LIN {X 0,Y 383.002,Z 302.767,A -85,B 0,C 180,E1 -11908.496,E2 -11908.496} C_VEL
LIN {X 0,Y 382.972,Z 302.776,A -85,B 0,C 180,E1 -11912.153,E2 -11912.153} C_VEL
LIN {X 0,Y 382.982,Z 302.775,A -85,B 0,C 180,E1 -11914.672,E2 -11914.672} C_VEL
LIN {X 0,Y 383.019,Z 302.772,A -85,B 0,C 180,E1 -11917.918,E2 -11917.918} C_VEL
LIN {X 0,Y 383.016,Z 302.775,A -85,B 0,C 180,E1 -11921.343,E2 -11921.343} C_VEL
LIN {X 0,Y 383.041,Z 302.775,A -85,B 0,C 180,E1 -11924.319,E2 -11924.319} C_VEL
LIN {X 0,Y 383.048,Z 302.775,A -85,B 0,C 180,E1 -11927.254,E2 -11927.254} C_VEL
LIN {X 0,Y 382.998,Z 302.778,A -85,B 0,C 180,E1 -11930.417,E2 -11930.417} C_VEL
LIN {X 0,Y 383.005,Z 302.774,A -85,B 0,C 180,E1 -11934.049,E2 -11934.049} C_VEL
LIN {X 0,Y 382.97,Z 302.788,A -85,B 0,C 180,E1 -11937.582,E2 -11937.582} C_VEL
LIN {X 0,Y 383.046,Z 302.81,A -85,B 0,C 180,E1 -11940.764,E2 -11940.764} C_VEL
LIN {X 0,Y 385.426,Z 313.551,A -85,B 0,C 180,E1 -11943.315,E2 -11943.315} C_VEL
LIN {X 0,Y 386.753,Z 320.992,A -85,B 0,C 180,E1 -11945.013,E2 -11945.013} C_VEL
LIN {X 0,Y 385.608,Z 335.888,A -85,B 0,C 180,E1 -11948.105,E2 -11948.105} C_VEL
LIN {X 0,Y 385.335,Z 339.604,A -85,B 0,C 180,E1 -11948.869,E2 -11948.869} C_VEL
LIN {X 0,Y 389.493,Z 364.024,A -85,B 0,C 180,E1 -11949.628,E2 -11949.628} C_VEL
LIN {X 0,Y 390.593,Z 373.139,A -85,B 0,C 180,E1 -11949.877,E2 -11949.877} C_VEL
LIN {X 0,Y 389.274,Z 448.59,A -85,B 0,C 180,E1 -11951.348,E2 -11951.348} C_VEL
LIN {X 0,Y 388.581,Z 462.418,A -85,B 0,C 180,E1 -11951.826,E2 -11951.826} C_VEL
LIN {X 0,Y 387.765,Z 474.887,A -85,B 0,C 180,E1 -11952.468,E2 -11952.468} C_VEL
LIN {X 0,Y 386.87,Z 486.049,A -85,B 0,C 180,E1 -11953.243,E2 -11953.243} C_VEL
LIN {X 0,Y 385.906,Z 497.675,A -85,B 0,C 180,E1 -11954.287,E2 -11954.287} C_VEL
LIN {X 0,Y 384.958,Z 508.376,A -85,B 0,C 180,E1 -11955.492,E2 -11955.492} C_VEL
LIN {X 0,Y 384.083,Z 517.643,A -85,B 0,C 180,E1 -11956.782,E2 -11956.782} C_VEL
LIN {X 0,Y 383.116,Z 526.789,A -85,B 0,C 180,E1 -11958.363,E2 -11958.363} C_VEL
LIN {X 0,Y 382.493,Z 534.178,A -85,B 0,C 180,E1 -11959.951,E2 -11959.951} C_VEL
LIN {X 0,Y 382.048,Z 540.112,A -85,B 0,C 180,E1 -11961.541,E2 -11961.541} C_VEL
LIN {X 0,Y 381.781,Z 544.795,A -85,B 0,C 180,E1 -11963.132,E2 -11963.132} C_VEL
LIN {X 0,Y 381.64,Z 548.367,A -85,B 0,C 180,E1 -11964.721,E2 -11964.721} C_VEL
LIN {X 0,Y 381.625,Z 550.176,A -85,B 0,C 180,E1 -11965.779,E2 -11965.779} C_VEL
LIN {X 0,Y 381.599,Z 552.53,A -85,B 0,C 180,E1 -11967.893,E2 -11967.893} C_VEL
LIN {X 0,Y 381.652,Z 553.116,A -85,B 0,C 180,E1 -11968.948,E2 -11968.948} C_VEL
LIN {X 0,Y 381.657,Z 553.261,A -85,B 0,C 180,E1 -11970.003,E2 -11970.003} C_VEL
LIN {X 0,Y 381.671,Z 553.002,A -85,B 0,C 180,E1 -11971.058,E2 -11971.058} C_VEL
LIN {X 0,Y 381.602,Z 552.348,A -85,B 0,C 180,E1 -11972.114,E2 -11972.114} C_VEL
LIN {X 0,Y 381.553,Z 551.297,A -85,B 0,C 180,E1 -11973.171,E2 -11973.171} C_VEL
LIN {X 0,Y 381.627,Z 549.792,A -85,B 0,C 180,E1 -11974.228,E2 -11974.228} C_VEL
LIN {X 0,Y 381.689,Z 546.003,A -85,B 0,C 180,E1 -11976.121,E2 -11976.121} C_VEL
LIN {X 0,Y 381.925,Z 540.955,A -85,B 0,C 180,E1 -11977.936,E2 -11977.936} C_VEL
LIN {X 0,Y 382.373,Z 534.098,A -85,B 0,C 180,E1 -11979.791,E2 -11979.791} C_VEL
LIN {X 0,Y 382.919,Z 526.632,A -85,B 0,C 180,E1 -11981.382,E2 -11981.382} C_VEL
LIN {X 0,Y 383.657,Z 519.027,A -85,B 0,C 180,E1 -11982.701,E2 -11982.701} C_VEL
LIN {X 0,Y 384.499,Z 509.401,A -85,B 0,C 180,E1 -11984.072,E2 -11984.072} C_VEL
LIN {X 0,Y 385.376,Z 498.26,A -85,B 0,C 180,E1 -11985.336,E2 -11985.336} C_VEL
LIN {X 0,Y 386.307,Z 486.607,A -85,B 0,C 180,E1 -11986.381,E2 -11986.381} C_VEL
LIN {X 0,Y 387.169,Z 474.246,A -85,B 0,C 180,E1 -11987.226,E2 -11987.226} C_VEL
LIN {X 0,Y 387.993,Z 461.29,A -85,B 0,C 180,E1 -11987.869,E2 -11987.869} C_VEL
LIN {X 0,Y 388.494,Z 448.766,A -85,B 0,C 180,E1 -11988.288,E2 -11988.288} C_VEL
LIN {X 0,Y 389.654,Z 371.374,A -85,B 0,C 180,E1 -11989.781,E2 -11989.781} C_VEL
LIN {X 0,Y 385.029,Z 340.715,A -85,B 0,C 180,E1 -11990.643,E2 -11990.643} C_VEL
LIN {X 0,Y 386.491,Z 322.694,A -85,B 0,C 180,E1 -11994.475,E2 -11994.475} C_VEL
LIN {X 0,Y 386.353,Z 318.928,A -85,B 0,C 180,E1 -11995.31,E2 -11995.31} C_VEL
LIN {X 0,Y 384.281,Z 308.331,A -85,B 0,C 180,E1 -11997.8,E2 -11997.8} C_VEL
LIN {X 0,Y 383.076,Z 302.77,A -85,B 0,C 180,E1 -11999.166,E2 -11999.166} C_VEL
LIN {X 0,Y 382.992,Z 302.777,A -85,B 0,C 180,E1 -12002.423,E2 -12002.423} C_VEL
LIN {X 0,Y 383.029,Z 302.773,A -85,B 0,C 180,E1 -12005.956,E2 -12005.956} C_VEL
LIN {X 0,Y 383.017,Z 302.771,A -85,B 0,C 180,E1 -12009.587,E2 -12009.587} C_VEL
LIN {X 0,Y 383.009,Z 302.774,A -85,B 0,C 180,E1 -12012.779,E2 -12012.779} C_VEL
LIN {X 0,Y 382.999,Z 302.774,A -85,B 0,C 180,E1 -12015.789,E2 -12015.789} C_VEL
LIN {X 0,Y 382.99,Z 302.778,A -85,B 0,C 180,E1 -12018.796,E2 -12018.796} C_VEL
LIN {X 0,Y 383.001,Z 302.774,A -85,B 0,C 180,E1 -12022.097,E2 -12022.097} C_VEL
LIN {X 0,Y 383.019,Z 302.771,A -85,B 0,C 180,E1 -12025.332,E2 -12025.332} C_VEL
LIN {X 0,Y 382.982,Z 302.778,A -85,B 0,C 180,E1 -12029.081,E2 -12029.081} C_VEL
LIN {X 0,Y 383.056,Z 302.771,A -85,B 0,C 180,E1 -12032.698,E2 -12032.698} C_VEL
LIN {X 0,Y 383.05,Z 302.772,A -85,B 0,C 180,E1 -12035.04,E2 -12035.04} C_VEL
LIN {X 0,Y 382.99,Z 302.776,A -85,B 0,C 180,E1 -12038.469,E2 -12038.469} C_VEL
LIN {X 0,Y 383.051,Z 302.767,A -85,B 0,C 180,E1 -12041.826,E2 -12041.826} C_VEL
LIN {X 0,Y 383.105,Z 302.767,A -85,B 0,C 180,E1 -12045.118,E2 -12045.118} C_VEL
LIN {X 0,Y 383.091,Z 302.761,A -85,B 0,C 180,E1 -12048.358,E2 -12048.358} C_VEL
LIN {X 0,Y 383.261,Z 302.741,A -85,B 0,C 180,E1 -12051.976,E2 -12051.976} C_VEL
LIN {X 0,Y 383.188,Z 302.75,A -85,B 0,C 180,E1 -12054.738,E2 -12054.738} C_VEL
LIN {X 0,Y 383.377,Z 302.728,A -85,B 0,C 180,E1 -12057.899,E2 -12057.899} C_VEL
LIN {X 0,Y 383.508,Z 302.711,A -85,B 0,C 180,E1 -12060,E2 -12060} C_VEL
LIN {X 0,Y 383.236,Z 302.746,A -85,B 0,C 180,E1 -12063.154,E2 -12063.154} C_VEL
LIN {X 0,Y 383.22,Z 302.745,A -85,B 0,C 180,E1 -12066.493,E2 -12066.493} C_VEL
LIN {X 0,Y 383.138,Z 302.76,A -85,B 0,C 180,E1 -12069.503,E2 -12069.503} C_VEL
LIN {X 0,Y 383.123,Z 302.761,A -85,B 0,C 180,E1 -12073.536,E2 -12073.536} C_VEL
LIN {X 0,Y 383.09,Z 302.761,A -85,B 0,C 180,E1 -12077.069,E2 -12077.069} C_VEL
LIN {X 0,Y 383.025,Z 302.77,A -85,B 0,C 180,E1 -12080.646,E2 -12080.646} C_VEL
LIN {X 0,Y 383.005,Z 302.776,A -85,B 0,C 180,E1 -12083.809,E2 -12083.809} C_VEL
LIN {X 0,Y 382.966,Z 302.777,A -85,B 0,C 180,E1 -12087.309,E2 -12087.309} C_VEL
LIN {X 0,Y 382.979,Z 302.776,A -85,B 0,C 180,E1 -12090.919,E2 -12090.919} C_VEL
LIN {X 0,Y 383.011,Z 302.774,A -85,B 0,C 180,E1 -12094.669,E2 -12094.669} C_VEL
LIN {X 0,Y 382.99,Z 302.776,A -85,B 0,C 180,E1 -12097.901,E2 -12097.901} C_VEL
LIN {X 0,Y 382.96,Z 302.778,A -85,B 0,C 180,E1 -12101.351,E2 -12101.351} C_VEL
LIN {X 0,Y 382.976,Z 302.78,A -85,B 0,C 180,E1 -12104.299,E2 -12104.299} C_VEL
LIN {X 0,Y 382.979,Z 302.776,A -85,B 0,C 180,E1 -12107.235,E2 -12107.235} C_VEL
LIN {X 0,Y 382.982,Z 302.779,A -85,B 0,C 180,E1 -12110.42,E2 -12110.42} C_VEL
LIN {X 0,Y 382.953,Z 302.778,A -85,B 0,C 180,E1 -12113.852,E2 -12113.852} C_VEL
LIN {X 0,Y 382.959,Z 302.782,A -85,B 0,C 180,E1 -12116.593,E2 -12116.593} C_VEL
LIN {X 0,Y 382.998,Z 302.773,A -85,B 0,C 180,E1 -12119.593,E2 -12119.593} C_VEL
LIN {X 0,Y 382.969,Z 302.78,A -85,B 0,C 180,E1 -12122.69,E2 -12122.69} C_VEL
LIN {X 0,Y 383.013,Z 302.771,A -85,B 0,C 180,E1 -12126.189,E2 -12126.189} C_VEL
LIN {X 0,Y 383.062,Z 302.767,A -85,B 0,C 180,E1 -12129.597,E2 -12129.597} C_VEL
LIN {X 0,Y 383.1,Z 302.764,A -85,B 0,C 180,E1 -12132.929,E2 -12132.929} C_VEL
LIN {X 0,Y 383.132,Z 302.756,A -85,B 0,C 180,E1 -12136.462,E2 -12136.462} C_VEL
LIN {X 0,Y 383.143,Z 302.755,A -85,B 0,C 180,E1 -12140.495,E2 -12140.495} C_VEL
LIN {X 0,Y 383.238,Z 302.748,A -85,B 0,C 180,E1 -12143.68,E2 -12143.68} C_VEL
LIN {X 0,Y 383.375,Z 302.729,A -85,B 0,C 180,E1 -12147.896,E2 -12147.896} C_VEL
LIN {X 0,Y 383.262,Z 302.741,A -85,B 0,C 180,E1 -12151.047,E2 -12151.047} C_VEL
LIN {X 0,Y 383.376,Z 302.728,A -85,B 0,C 180,E1 -12152.098,E2 -12152.098} C_VEL
LIN {X 0,Y 383.235,Z 302.749,A -85,B 0,C 180,E1 -12156.313,E2 -12156.313} C_VEL
LIN {X 0,Y 383.193,Z 302.89,A -85,B 0,C 180,E1 -12158.566,E2 -12158.566} C_VEL
LIN {X 0,Y 385.187,Z 313.862,A -85,B 0,C 180,E1 -12161.44,E2 -12161.44} C_VEL
LIN {X 0,Y 388.871,Z 330.52,A -85,B 0,C 180,E1 -12161.975,E2 -12161.975} C_VEL
LIN {X 0,Y 390.045,Z 336.622,A -85,B 0,C 180,E1 -12162.156,E2 -12162.156} C_VEL
LIN {X 0,Y 388.665,Z 421.372,A -85,B 0,C 180,E1 -12163.791,E2 -12163.791} C_VEL
LIN {X 0,Y 388.202,Z 435.09,A -85,B 0,C 180,E1 -12164.276,E2 -12164.276} C_VEL
LIN {X 0,Y 387.769,Z 443.992,A -85,B 0,C 180,E1 -12164.72,E2 -12164.72} C_VEL
LIN {X 0,Y 386.844,Z 449.578,A -85,B 0,C 180,E1 -12165.029,E2 -12165.029} C_VEL
LIN {X 0,Y 383.446,Z 458.33,A -85,B 0,C 180,E1 -12165.533,E2 -12165.533} C_VEL
LIN {X 0,Y 380.038,Z 466.639,A -85,B 0,C 180,E1 -12166.14,E2 -12166.14} C_VEL
LIN {X 0,Y 379.082,Z 471.479,A -85,B 0,C 180,E1 -12166.602,E2 -12166.602} C_VEL
LIN {X 0,Y 378.117,Z 482.102,A -85,B 0,C 180,E1 -12167.854,E2 -12167.854} C_VEL
LIN {X 0,Y 377.244,Z 491.895,A -85,B 0,C 180,E1 -12169.305,E2 -12169.305} C_VEL
LIN {X 0,Y 376.543,Z 499.898,A -85,B 0,C 180,E1 -12170.765,E2 -12170.765} C_VEL
LIN {X 0,Y 375.905,Z 506.51,A -85,B 0,C 180,E1 -12172.241,E2 -12172.241} C_VEL
LIN {X 0,Y 375.413,Z 512.368,A -85,B 0,C 180,E1 -12173.863,E2 -12173.863} C_VEL
LIN {X 0,Y 374.981,Z 517.914,A -85,B 0,C 180,E1 -12175.89,E2 -12175.89} C_VEL
LIN {X 0,Y 374.593,Z 521.91,A -85,B 0,C 180,E1 -12177.966,E2 -12177.966} C_VEL
LIN {X 0,Y 374.449,Z 523.478,A -85,B 0,C 180,E1 -12179.202,E2 -12179.202} C_VEL
LIN {X 0,Y 374.394,Z 524.558,A -85,B 0,C 180,E1 -12180.447,E2 -12180.447} C_VEL
LIN {X 0,Y 374.34,Z 525.133,A -85,B 0,C 180,E1 -12182.344,E2 -12182.344} C_VEL
LIN {X 0,Y 374.422,Z 524.402,A -85,B 0,C 180,E1 -12184.321,E2 -12184.321} C_VEL
LIN {X 0,Y 374.645,Z 522.422,A -85,B 0,C 180,E1 -12186.231,E2 -12186.231} C_VEL
LIN {X 0,Y 374.984,Z 519.015,A -85,B 0,C 180,E1 -12188.198,E2 -12188.198} C_VEL
LIN {X 0,Y 375.356,Z 514.94,A -85,B 0,C 180,E1 -12189.855,E2 -12189.855} C_VEL
LIN {X 0,Y 375.921,Z 509.32,A -85,B 0,C 180,E1 -12191.598,E2 -12191.598} C_VEL
LIN {X 0,Y 376.685,Z 502.286,A -85,B 0,C 180,E1 -12193.311,E2 -12193.311} C_VEL
LIN {X 0,Y 377.463,Z 495.497,A -85,B 0,C 180,E1 -12194.649,E2 -12194.649} C_VEL
LIN {X 0,Y 378.359,Z 487.043,A -85,B 0,C 180,E1 -12196.027,E2 -12196.027} C_VEL
LIN {X 0,Y 379.359,Z 477.432,A -85,B 0,C 180,E1 -12197.302,E2 -12197.302} C_VEL
LIN {X 0,Y 380.255,Z 467.275,A -85,B 0,C 180,E1 -12198.39,E2 -12198.39} C_VEL
LIN {X 0,Y 381.225,Z 455.072,A -85,B 0,C 180,E1 -12199.423,E2 -12199.423} C_VEL
LIN {X 0,Y 382.078,Z 442.777,A -85,B 0,C 180,E1 -12200.208,E2 -12200.208} C_VEL
LIN {X 0,Y 382.618,Z 429.417,A -85,B 0,C 180,E1 -12200.815,E2 -12200.815} C_VEL
LIN {X 0,Y 383.072,Z 416.771,A -85,B 0,C 180,E1 -12201.171,E2 -12201.171} C_VEL
LIN {X 0,Y 384.452,Z 337.546,A -85,B 0,C 180,E1 -12202.732,E2 -12202.732} C_VEL
LIN {X 0,Y 380.635,Z 320.427,A -85,B 0,C 180,E1 -12203.339,E2 -12203.339} C_VEL
LIN {X 0,Y 378.249,Z 314.133,A -85,B 0,C 180,E1 -12203.642,E2 -12203.642} C_VEL
LIN {X 0,Y 375.961,Z 303.656,A -85,B 0,C 180,E1 -12206.211,E2 -12206.211} C_VEL
LIN {X 0,Y 375.928,Z 303.659,A -85,B 0,C 180,E1 -12209.684,E2 -12209.684} C_VEL
LIN {X 0,Y 375.956,Z 303.66,A -85,B 0,C 180,E1 -12212.138,E2 -12212.138} C_VEL
LIN {X 0,Y 375.964,Z 303.659,A -85,B 0,C 180,E1 -12214.536,E2 -12214.536} C_VEL
LIN {X 0,Y 375.914,Z 303.666,A -85,B 0,C 180,E1 -12218.043,E2 -12218.043} C_VEL
LIN {X 0,Y 375.962,Z 303.652,A -85,B 0,C 180,E1 -12221.471,E2 -12221.471} C_VEL
LIN {X 0,Y 376.01,Z 303.65,A -85,B 0,C 180,E1 -12224.83,E2 -12224.83} C_VEL
LIN {X 0,Y 376.001,Z 303.648,A -85,B 0,C 180,E1 -12228.135,E2 -12228.135} C_VEL
LIN {X 0,Y 376.171,Z 303.625,A -85,B 0,C 180,E1 -12231.918,E2 -12231.918} C_VEL
LIN {X 0,Y 376.12,Z 303.636,A -85,B 0,C 180,E1 -12234.639,E2 -12234.639} C_VEL
LIN {X 0,Y 376.305,Z 303.608,A -85,B 0,C 180,E1 -12237.859,E2 -12237.859} C_VEL
LIN {X 0,Y 376.439,Z 303.584,A -85,B 0,C 180,E1 -12240,E2 -12240} C_VEL
LIN {X 0,Y 376.147,Z 303.624,A -85,B 0,C 180,E1 -12243.213,E2 -12243.213} C_VEL
LIN {X 0,Y 376.193,Z 303.623,A -85,B 0,C 180,E1 -12246.436,E2 -12246.436} C_VEL
LIN {X 0,Y 376.077,Z 303.638,A -85,B 0,C 180,E1 -12249.683,E2 -12249.683} C_VEL
LIN {X 0,Y 376.043,Z 303.642,A -85,B 0,C 180,E1 -12253.659,E2 -12253.659} C_VEL
LIN {X 0,Y 376,Z 303.647,A -85,B 0,C 180,E1 -12257.61,E2 -12257.61} C_VEL
LIN {X 0,Y 375.967,Z 303.643,A -85,B 0,C 180,E1 -12260.848,E2 -12260.848} C_VEL
LIN {X 0,Y 375.958,Z 303.643,A -85,B 0,C 180,E1 -12264.284,E2 -12264.284} C_VEL
LIN {X 0,Y 375.979,Z 303.647,A -85,B 0,C 180,E1 -12266.655,E2 -12266.655} C_VEL
LIN {X 0,Y 375.933,Z 303.651,A -85,B 0,C 180,E1 -12269.082,E2 -12269.082} C_VEL
LIN {X 0,Y 375.912,Z 303.656,A -85,B 0,C 180,E1 -12272.832,E2 -12272.832} C_VEL
LIN {X 0,Y 375.976,Z 303.65,A -85,B 0,C 180,E1 -12276.518,E2 -12276.518} C_VEL
LIN {X 0,Y 375.976,Z 303.653,A -85,B 0,C 180,E1 -12279.979,E2 -12279.979} C_VEL
LIN {X 0,Y 375.971,Z 303.655,A -85,B 0,C 180,E1 -12283.76,E2 -12283.76} C_VEL
LIN {X 0,Y 375.971,Z 303.655,A -85,B 0,C 180,E1 -12286.805,E2 -12286.805} C_VEL
LIN {X 0,Y 375.975,Z 303.654,A -85,B 0,C 180,E1 -12290.032,E2 -12290.032} C_VEL
LIN {X 0,Y 375.944,Z 303.654,A -85,B 0,C 180,E1 -12293.5,E2 -12293.5} C_VEL
LIN {X 0,Y 375.94,Z 303.659,A -85,B 0,C 180,E1 -12295.893,E2 -12295.893} C_VEL
LIN {X 0,Y 375.953,Z 303.663,A -85,B 0,C 180,E1 -12299.693,E2 -12299.693} C_VEL
LIN {X 0,Y 375.972,Z 303.722,A -85,B 0,C 180,E1 -12300.39,E2 -12300.39} C_VEL
LIN {X 0,Y 378.629,Z 315.49,A -85,B 0,C 180,E1 -12303.255,E2 -12303.255} C_VEL
LIN {X 0,Y 379.852,Z 322.212,A -85,B 0,C 180,E1 -12304.821,E2 -12304.821} C_VEL
LIN {X 0,Y 378.688,Z 337.055,A -85,B 0,C 180,E1 -12307.96,E2 -12307.96} C_VEL
LIN {X 0,Y 378.5,Z 339.273,A -85,B 0,C 180,E1 -12308.424,E2 -12308.424} C_VEL
LIN {X 0,Y 382.634,Z 363.105,A -85,B 0,C 180,E1 -12309.197,E2 -12309.197} C_VEL
LIN {X 0,Y 384.003,Z 372.756,A -85,B 0,C 180,E1 -12309.482,E2 -12309.482} C_VEL
LIN {X 0,Y 382.629,Z 448.146,A -85,B 0,C 180,E1 -12310.977,E2 -12310.977} C_VEL
LIN {X 0,Y 381.916,Z 462.023,A -85,B 0,C 180,E1 -12311.462,E2 -12311.462} C_VEL
LIN {X 0,Y 381.014,Z 475.057,A -85,B 0,C 180,E1 -12312.147,E2 -12312.147} C_VEL
LIN {X 0,Y 379.959,Z 487.685,A -85,B 0,C 180,E1 -12313.068,E2 -12313.068} C_VEL
LIN {X 0,Y 378.967,Z 498.961,A -85,B 0,C 180,E1 -12314.13,E2 -12314.13} C_VEL
LIN {X 0,Y 377.935,Z 509.706,A -85,B 0,C 180,E1 -12315.406,E2 -12315.406} C_VEL
LIN {X 0,Y 376.987,Z 519.159,A -85,B 0,C 180,E1 -12316.803,E2 -12316.803} C_VEL
LIN {X 0,Y 375.989,Z 527.997,A -85,B 0,C 180,E1 -12318.412,E2 -12318.412} C_VEL
LIN {X 0,Y 375.381,Z 535.076,A -85,B 0,C 180,E1 -12320.031,E2 -12320.031} C_VEL
LIN {X 0,Y 374.877,Z 541.577,A -85,B 0,C 180,E1 -12321.921,E2 -12321.921} C_VEL
LIN {X 0,Y 374.628,Z 545.863,A -85,B 0,C 180,E1 -12323.541,E2 -12323.541} C_VEL
LIN {X 0,Y 374.551,Z 548.144,A -85,B 0,C 180,E1 -12324.621,E2 -12324.621} C_VEL
LIN {X 0,Y 374.55,Z 549.94,A -85,B 0,C 180,E1 -12325.699,E2 -12325.699} C_VEL
LIN {X 0,Y 374.497,Z 552.282,A -85,B 0,C 180,E1 -12327.853,E2 -12327.853} C_VEL
LIN {X 0,Y 374.567,Z 552.859,A -85,B 0,C 180,E1 -12328.928,E2 -12328.928} C_VEL
LIN {X 0,Y 374.59,Z 552.993,A -85,B 0,C 180,E1 -12330.003,E2 -12330.003} C_VEL
LIN {X 0,Y 374.584,Z 552.725,A -85,B 0,C 180,E1 -12331.078,E2 -12331.078} C_VEL
LIN {X 0,Y 374.502,Z 552.063,A -85,B 0,C 180,E1 -12332.154,E2 -12332.154} C_VEL
LIN {X 0,Y 374.467,Z 551.002,A -85,B 0,C 180,E1 -12333.231,E2 -12333.231} C_VEL
LIN {X 0,Y 374.553,Z 549.484,A -85,B 0,C 180,E1 -12334.308,E2 -12334.308} C_VEL
LIN {X 0,Y 374.585,Z 546.066,A -85,B 0,C 180,E1 -12336.069,E2 -12336.069} C_VEL
LIN {X 0,Y 374.774,Z 542.239,A -85,B 0,C 180,E1 -12337.546,E2 -12337.546} C_VEL
LIN {X 0,Y 375.162,Z 535.869,A -85,B 0,C 180,E1 -12339.437,E2 -12339.437} C_VEL
LIN {X 0,Y 375.701,Z 528.925,A -85,B 0,C 180,E1 -12341.057,E2 -12341.057} C_VEL
LIN {X 0,Y 376.547,Z 520.229,A -85,B 0,C 180,E1 -12342.671,E2 -12342.671} C_VEL
LIN {X 0,Y 377.352,Z 511.3,A -85,B 0,C 180,E1 -12344.014,E2 -12344.014} C_VEL
LIN {X 0,Y 378.275,Z 500.298,A -85,B 0,C 180,E1 -12345.355,E2 -12345.355} C_VEL
LIN {X 0,Y 379.196,Z 489.168,A -85,B 0,C 180,E1 -12346.42,E2 -12346.42} C_VEL
LIN {X 0,Y 380.191,Z 476.715,A -85,B 0,C 180,E1 -12347.345,E2 -12347.345} C_VEL
LIN {X 0,Y 380.932,Z 464.872,A -85,B 0,C 180,E1 -12348.003,E2 -12348.003} C_VEL
LIN {X 0,Y 381.585,Z 452.019,A -85,B 0,C 180,E1 -12348.492,E2 -12348.492} C_VEL
LIN {X 0,Y 382.001,Z 432.44,A -85,B 0,C 180,E1 -12348.923,E2 -12348.923} C_VEL
LIN {X 0,Y 382.867,Z 371.861,A -85,B 0,C 180,E1 -12350.103,E2 -12350.103} C_VEL
LIN {X 0,Y 378.139,Z 340.495,A -85,B 0,C 180,E1 -12350.999,E2 -12350.999} C_VEL
LIN {X 0,Y 379.505,Z 324.471,A -85,B 0,C 180,E1 -12354.471,E2 -12354.471} C_VEL
LIN {X 0,Y 379.555,Z 321.157,A -85,B 0,C 180,E1 -12355.208,E2 -12355.208} C_VEL
LIN {X 0,Y 377.277,Z 309.402,A -85,B 0,C 180,E1 -12358.019,E2 -12358.019} C_VEL
LIN {X 0,Y 375.995,Z 303.651,A -85,B 0,C 180,E1 -12359.462,E2 -12359.462} C_VEL
LIN {X 0,Y 375.955,Z 303.651,A -85,B 0,C 180,E1 -12362.83,E2 -12362.83} C_VEL
LIN {X 0,Y 375.962,Z 303.65,A -85,B 0,C 180,E1 -12365.416,E2 -12365.416} C_VEL
LIN {X 0,Y 375.976,Z 303.655,A -85,B 0,C 180,E1 -12368.27,E2 -12368.27} C_VEL
LIN {X 0,Y 375.937,Z 303.653,A -85,B 0,C 180,E1 -12371.601,E2 -12371.601} C_VEL
LIN {X 0,Y 375.929,Z 303.654,A -85,B 0,C 180,E1 -12375.269,E2 -12375.269} C_VEL
LIN {X 0,Y 375.937,Z 303.659,A -85,B 0,C 180,E1 -12378.4,E2 -12378.4} C_VEL
LIN {X 0,Y 375.975,Z 303.648,A -85,B 0,C 180,E1 -12381.73,E2 -12381.73} C_VEL
LIN {X 0,Y 375.981,Z 303.648,A -85,B 0,C 180,E1 -12385.333,E2 -12385.333} C_VEL
LIN {X 0,Y 375.957,Z 303.654,A -85,B 0,C 180,E1 -12388.438,E2 -12388.438} C_VEL
LIN {X 0,Y 375.982,Z 303.648,A -85,B 0,C 180,E1 -12392.14,E2 -12392.14} C_VEL
LIN {X 0,Y 376.005,Z 303.647,A -85,B 0,C 180,E1 -12394.539,E2 -12394.539} C_VEL
LIN {X 0,Y 375.956,Z 303.65,A -85,B 0,C 180,E1 -12398.045,E2 -12398.045} C_VEL
LIN {X 0,Y 376.001,Z 303.647,A -85,B 0,C 180,E1 -12401.473,E2 -12401.473} C_VEL
LIN {X 0,Y 376.054,Z 303.642,A -85,B 0,C 180,E1 -12404.832,E2 -12404.832} C_VEL
LIN {X 0,Y 376.043,Z 303.639,A -85,B 0,C 180,E1 -12408.136,E2 -12408.136} C_VEL
LIN {X 0,Y 376.216,Z 303.619,A -85,B 0,C 180,E1 -12411.919,E2 -12411.919} C_VEL
LIN {X 0,Y 376.161,Z 303.625,A -85,B 0,C 180,E1 -12414.64,E2 -12414.64} C_VEL
LIN {X 0,Y 376.344,Z 303.604,A -85,B 0,C 180,E1 -12417.86,E2 -12417.86} C_VEL
LIN {X 0,Y 376.478,Z 303.587,A -85,B 0,C 180,E1 -12420,E2 -12420} C_VEL
LIN {X 0,Y 376.344,Z 303.603,A -85,B 0,C 180,E1 -12422.14,E2 -12422.14} C_VEL
LIN {X 0,Y 376.191,Z 303.621,A -85,B 0,C 180,E1 -12426.478,E2 -12426.478} C_VEL
LIN {X 0,Y 376.108,Z 303.638,A -85,B 0,C 180,E1 -12429.682,E2 -12429.682} C_VEL
LIN {X 0,Y 376.087,Z 303.639,A -85,B 0,C 180,E1 -12433.657,E2 -12433.657} C_VEL
LIN {X 0,Y 376.029,Z 303.643,A -85,B 0,C 180,E1 -12437.4,E2 -12437.4} C_VEL
LIN {X 0,Y 375.978,Z 303.647,A -85,B 0,C 180,E1 -12440.832,E2 -12440.832} C_VEL
LIN {X 0,Y 375.932,Z 303.658,A -85,B 0,C 180,E1 -12444.286,E2 -12444.286} C_VEL
LIN {X 0,Y 375.909,Z 303.657,A -85,B 0,C 180,E1 -12446.661,E2 -12446.661} C_VEL
LIN {X 0,Y 375.912,Z 303.656,A -85,B 0,C 180,E1 -12449.084,E2 -12449.084} C_VEL
LIN {X 0,Y 375.936,Z 303.653,A -85,B 0,C 180,E1 -12451.564,E2 -12451.564} C_VEL
LIN {X 0,Y 375.974,Z 303.651,A -85,B 0,C 180,E1 -12454.666,E2 -12454.666} C_VEL
LIN {X 0,Y 375.931,Z 303.659,A -85,B 0,C 180,E1 -12458.262,E2 -12458.262} C_VEL
LIN {X 0,Y 375.913,Z 303.655,A -85,B 0,C 180,E1 -12461.596,E2 -12461.596} C_VEL
LIN {X 0,Y 375.904,Z 303.661,A -85,B 0,C 180,E1 -12464.727,E2 -12464.727} C_VEL
LIN {X 0,Y 375.912,Z 303.66,A -85,B 0,C 180,E1 -12468.403,E2 -12468.403} C_VEL
LIN {X 0,Y 375.948,Z 303.651,A -85,B 0,C 180,E1 -12471.908,E2 -12471.908} C_VEL
LIN {X 0,Y 375.929,Z 303.655,A -85,B 0,C 180,E1 -12475.344,E2 -12475.344} C_VEL
LIN {X 0,Y 375.934,Z 303.655,A -85,B 0,C 180,E1 -12478.434,E2 -12478.434} C_VEL
LIN {X 0,Y 375.952,Z 303.652,A -85,B 0,C 180,E1 -12481.476,E2 -12481.476} C_VEL
LIN {X 0,Y 375.953,Z 303.652,A -85,B 0,C 180,E1 -12484.533,E2 -12484.533} C_VEL
LIN {X 0,Y 375.96,Z 303.649,A -85,B 0,C 180,E1 -12488.043,E2 -12488.043} C_VEL
LIN {X 0,Y 376.008,Z 303.647,A -85,B 0,C 180,E1 -12491.471,E2 -12491.471} C_VEL
LIN {X 0,Y 376.061,Z 303.639,A -85,B 0,C 180,E1 -12494.83,E2 -12494.83} C_VEL
LIN {X 0,Y 376.051,Z 303.638,A -85,B 0,C 180,E1 -12498.134,E2 -12498.134} C_VEL
LIN {X 0,Y 376.191,Z 303.622,A -85,B 0,C 180,E1 -12501.952,E2 -12501.952} C_VEL
LIN {X 0,Y 376.147,Z 303.626,A -85,B 0,C 180,E1 -12504.636,E2 -12504.636} C_VEL
LIN {X 0,Y 376.34,Z 303.606,A -85,B 0,C 180,E1 -12507.856,E2 -12507.856} C_VEL
LIN {X 0,Y 376.233,Z 303.617,A -85,B 0,C 180,E1 -12511.067,E2 -12511.067} C_VEL
LIN {X 0,Y 376.34,Z 303.604,A -85,B 0,C 180,E1 -12512.137,E2 -12512.137} C_VEL
LIN {X 0,Y 376.192,Z 303.626,A -85,B 0,C 180,E1 -12516.432,E2 -12516.432} C_VEL
LIN {X 0,Y 376.178,Z 303.786,A -85,B 0,C 180,E1 -12518.309,E2 -12518.309} C_VEL
LIN {X 0,Y 378.101,Z 314.257,A -85,B 0,C 180,E1 -12521.08,E2 -12521.08} C_VEL
LIN {X 0,Y 380.338,Z 322.774,A -85,B 0,C 180,E1 -12521.376,E2 -12521.376} C_VEL
LIN {X 0,Y 383.34,Z 338.495,A -85,B 0,C 180,E1 -12521.853,E2 -12521.853} C_VEL
LIN {X 0,Y 381.897,Z 421.344,A -85,B 0,C 180,E1 -12523.477,E2 -12523.477} C_VEL
LIN {X 0,Y 381.421,Z 434.845,A -85,B 0,C 180,E1 -12523.957,E2 -12523.957} C_VEL
LIN {X 0,Y 380.809,Z 447.559,A -85,B 0,C 180,E1 -12524.627,E2 -12524.627} C_VEL
LIN {X 0,Y 380.071,Z 459.028,A -85,B 0,C 180,E1 -12525.447,E2 -12525.447} C_VEL
LIN {X 0,Y 379.105,Z 471.034,A -85,B 0,C 180,E1 -12526.556,E2 -12526.556} C_VEL
LIN {X 0,Y 379.082,Z 471.479,A -85,B 0,C 180,E1 -12526.602,E2 -12526.602} C_VEL
LIN {X 0,Y 378.118,Z 476.284,A -85,B 0,C 180,E1 -12527.103,E2 -12527.103} C_VEL
LIN {X 0,Y 374.622,Z 483.802,A -85,B 0,C 180,E1 -12527.936,E2 -12527.936} C_VEL
LIN {X 0,Y 371.061,Z 490.776,A -85,B 0,C 180,E1 -12528.876,E2 -12528.876} C_VEL
LIN {X 0,Y 370.014,Z 494.728,A -85,B 0,C 180,E1 -12529.537,E2 -12529.537} C_VEL
LIN {X 0,Y 369.257,Z 503.014,A -85,B 0,C 180,E1 -12531.195,E2 -12531.195} C_VEL
LIN {X 0,Y 368.612,Z 510.198,A -85,B 0,C 180,E1 -12533.002,E2 -12533.002} C_VEL
LIN {X 0,Y 368.115,Z 515.785,A -85,B 0,C 180,E1 -12534.83,E2 -12534.83} C_VEL
LIN {X 0,Y 367.744,Z 520.033,A -85,B 0,C 180,E1 -12536.68,E2 -12536.68} C_VEL
LIN {X 0,Y 367.426,Z 523.045,A -85,B 0,C 180,E1 -12538.561,E2 -12538.561} C_VEL
LIN {X 0,Y 367.287,Z 524.895,A -85,B 0,C 180,E1 -12540.563,E2 -12540.563} C_VEL
LIN {X 0,Y 367.252,Z 525.365,A -85,B 0,C 180,E1 -12542.646,E2 -12542.646} C_VEL
LIN {X 0,Y 367.369,Z 524.484,A -85,B 0,C 180,E1 -12544.652,E2 -12544.652} C_VEL
LIN {X 0,Y 367.612,Z 522.369,A -85,B 0,C 180,E1 -12546.586,E2 -12546.586} C_VEL
LIN {X 0,Y 367.943,Z 519.056,A -85,B 0,C 180,E1 -12548.451,E2 -12548.451} C_VEL
LIN {X 0,Y 368.464,Z 514.088,A -85,B 0,C 180,E1 -12550.421,E2 -12550.421} C_VEL
LIN {X 0,Y 369.116,Z 507.965,A -85,B 0,C 180,E1 -12552.258,E2 -12552.258} C_VEL
LIN {X 0,Y 369.848,Z 501.589,A -85,B 0,C 180,E1 -12553.772,E2 -12553.772} C_VEL
LIN {X 0,Y 370.771,Z 493.971,A -85,B 0,C 180,E1 -12555.244,E2 -12555.244} C_VEL
LIN {X 0,Y 371.807,Z 484.763,A -85,B 0,C 180,E1 -12556.688,E2 -12556.688} C_VEL
LIN {X 0,Y 372.746,Z 475.071,A -85,B 0,C 180,E1 -12557.927,E2 -12557.927} C_VEL
LIN {X 0,Y 373.892,Z 463.81,A -85,B 0,C 180,E1 -12559.075,E2 -12559.075} C_VEL
LIN {X 0,Y 374.801,Z 452.082,A -85,B 0,C 180,E1 -12560.006,E2 -12560.006} C_VEL
LIN {X 0,Y 375.552,Z 439.813,A -85,B 0,C 180,E1 -12560.743,E2 -12560.743} C_VEL
LIN {X 0,Y 376.139,Z 427.194,A -85,B 0,C 180,E1 -12561.277,E2 -12561.277} C_VEL
LIN {X 0,Y 376.567,Z 411.448,A -85,B 0,C 180,E1 -12561.664,E2 -12561.664} C_VEL
LIN {X 0,Y 377.899,Z 338.583,A -85,B 0,C 180,E1 -12563.131,E2 -12563.131} C_VEL
LIN {X 0,Y 374.404,Z 322.818,A -85,B 0,C 180,E1 -12563.706,E2 -12563.706} C_VEL
LIN {X 0,Y 371.114,Z 314.42,A -85,B 0,C 180,E1 -12564.125,E2 -12564.125} C_VEL
LIN {X 0,Y 368.901,Z 304.536,A -85,B 0,C 180,E1 -12566.646,E2 -12566.646} C_VEL
LIN {X 0,Y 368.882,Z 304.539,A -85,B 0,C 180,E1 -12570.307,E2 -12570.307} C_VEL
LIN {X 0,Y 368.94,Z 304.533,A -85,B 0,C 180,E1 -12573.532,E2 -12573.532} C_VEL
LIN {X 0,Y 368.923,Z 304.536,A -85,B 0,C 180,E1 -12576.418,E2 -12576.418} C_VEL
LIN {X 0,Y 368.885,Z 304.539,A -85,B 0,C 180,E1 -12579.944,E2 -12579.944} C_VEL
LIN {X 0,Y 368.928,Z 304.528,A -85,B 0,C 180,E1 -12583.396,E2 -12583.396} C_VEL
LIN {X 0,Y 369.01,Z 304.518,A -85,B 0,C 180,E1 -12586.788,E2 -12586.788} C_VEL
LIN {X 0,Y 369.019,Z 304.514,A -85,B 0,C 180,E1 -12590.13,E2 -12590.13} C_VEL
LIN {X 0,Y 369.151,Z 304.499,A -85,B 0,C 180,E1 -12593.441,E2 -12593.441} C_VEL
LIN {X 0,Y 369.27,Z 304.484,A -85,B 0,C 180,E1 -12597.819,E2 -12597.819} C_VEL
LIN {X 0,Y 369.409,Z 304.46,A -85,B 0,C 180,E1 -12600,E2 -12600} C_VEL
LIN {X 0,Y 369.271,Z 304.484,A -85,B 0,C 180,E1 -12602.181,E2 -12602.181} C_VEL
LIN {X 0,Y 369.154,Z 304.501,A -85,B 0,C 180,E1 -12606.559,E2 -12606.559} C_VEL
LIN {X 0,Y 369.076,Z 304.506,A -85,B 0,C 180,E1 -12608.762,E2 -12608.762} C_VEL
LIN {X 0,Y 368.966,Z 304.515,A -85,B 0,C 180,E1 -12612.095,E2 -12612.095} C_VEL
LIN {X 0,Y 368.954,Z 304.52,A -85,B 0,C 180,E1 -12615.467,E2 -12615.467} C_VEL
LIN {X 0,Y 368.948,Z 304.526,A -85,B 0,C 180,E1 -12618.895,E2 -12618.895} C_VEL
LIN {X 0,Y 368.93,Z 304.524,A -85,B 0,C 180,E1 -12622.395,E2 -12622.395} C_VEL
LIN {X 0,Y 368.959,Z 304.522,A -85,B 0,C 180,E1 -12625.983,E2 -12625.983} C_VEL
LIN {X 0,Y 368.923,Z 304.522,A -85,B 0,C 180,E1 -12628.815,E2 -12628.815} C_VEL
LIN {X 0,Y 368.861,Z 304.533,A -85,B 0,C 180,E1 -12632.242,E2 -12632.242} C_VEL
LIN {X 0,Y 368.894,Z 304.531,A -85,B 0,C 180,E1 -12635.005,E2 -12635.005} C_VEL
LIN {X 0,Y 368.945,Z 304.524,A -85,B 0,C 180,E1 -12638.658,E2 -12638.658} C_VEL
LIN {X 0,Y 368.912,Z 304.536,A -85,B 0,C 180,E1 -12642.024,E2 -12642.024} C_VEL
LIN {X 0,Y 368.962,Z 304.53,A -85,B 0,C 180,E1 -12645.197,E2 -12645.197} C_VEL
LIN {X 0,Y 368.915,Z 304.534,A -85,B 0,C 180,E1 -12648.19,E2 -12648.19} C_VEL
LIN {X 0,Y 368.89,Z 304.537,A -85,B 0,C 180,E1 -12651.364,E2 -12651.364} C_VEL
LIN {X 0,Y 368.916,Z 304.534,A -85,B 0,C 180,E1 -12655.151,E2 -12655.151} C_VEL
LIN {X 0,Y 368.912,Z 304.538,A -85,B 0,C 180,E1 -12659.051,E2 -12659.051} C_VEL
LIN {X 0,Y 368.921,Z 304.643,A -85,B 0,C 180,E1 -12660.002,E2 -12660.002} C_VEL
LIN {X 0,Y 371.462,Z 315.766,A -85,B 0,C 180,E1 -12662.777,E2 -12662.777} C_VEL
LIN {X 0,Y 372.977,Z 324.032,A -85,B 0,C 180,E1 -12664.752,E2 -12664.752} C_VEL
LIN {X 0,Y 371.716,Z 338.619,A -85,B 0,C 180,E1 -12667.887,E2 -12667.887} C_VEL
LIN {X 0,Y 371.739,Z 339.318,A -85,B 0,C 180,E1 -12667.979,E2 -12667.979} C_VEL
LIN {X 0,Y 375.646,Z 360.977,A -85,B 0,C 180,E1 -12668.709,E2 -12668.709} C_VEL
LIN {X 0,Y 377.391,Z 374.932,A -85,B 0,C 180,E1 -12669.121,E2 -12669.121} C_VEL
LIN {X 0,Y 375.966,Z 448.82,A -85,B 0,C 180,E1 -12670.627,E2 -12670.627} C_VEL
LIN {X 0,Y 375.218,Z 462.38,A -85,B 0,C 180,E1 -12671.119,E2 -12671.119} C_VEL
LIN {X 0,Y 374.283,Z 475.204,A -85,B 0,C 180,E1 -12671.815,E2 -12671.815} C_VEL
LIN {X 0,Y 373.179,Z 487.74,A -85,B 0,C 180,E1 -12672.75,E2 -12672.75} C_VEL
LIN {X 0,Y 372.116,Z 498.957,A -85,B 0,C 180,E1 -12673.83,E2 -12673.83} C_VEL
LIN {X 0,Y 371.137,Z 508.438,A -85,B 0,C 180,E1 -12674.963,E2 -12674.963} C_VEL
LIN {X 0,Y 370.217,Z 517.417,A -85,B 0,C 180,E1 -12676.278,E2 -12676.278} C_VEL
LIN {X 0,Y 369.204,Z 526.504,A -85,B 0,C 180,E1 -12677.918,E2 -12677.918} C_VEL
LIN {X 0,Y 368.47,Z 533.844,A -85,B 0,C 180,E1 -12679.565,E2 -12679.565} C_VEL
LIN {X 0,Y 367.968,Z 539.732,A -85,B 0,C 180,E1 -12681.215,E2 -12681.215} C_VEL
LIN {X 0,Y 367.657,Z 544.377,A -85,B 0,C 180,E1 -12682.867,E2 -12682.867} C_VEL
LIN {X 0,Y 367.464,Z 547.92,A -85,B 0,C 180,E1 -12684.516,E2 -12684.516} C_VEL
LIN {X 0,Y 367.455,Z 549.705,A -85,B 0,C 180,E1 -12685.616,E2 -12685.616} C_VEL
LIN {X 0,Y 367.397,Z 552.034,A -85,B 0,C 180,E1 -12687.811,E2 -12687.811} C_VEL
LIN {X 0,Y 367.468,Z 552.6,A -85,B 0,C 180,E1 -12688.908,E2 -12688.908} C_VEL
LIN {X 0,Y 367.506,Z 552.724,A -85,B 0,C 180,E1 -12690.004,E2 -12690.004} C_VEL
LIN {X 0,Y 367.485,Z 552.449,A -85,B 0,C 180,E1 -12691.099,E2 -12691.099} C_VEL
LIN {X 0,Y 367.402,Z 551.779,A -85,B 0,C 180,E1 -12692.196,E2 -12692.196} C_VEL
LIN {X 0,Y 367.385,Z 550.706,A -85,B 0,C 180,E1 -12693.293,E2 -12693.293} C_VEL
LIN {X 0,Y 367.458,Z 549.174,A -85,B 0,C 180,E1 -12694.391,E2 -12694.391} C_VEL
LIN {X 0,Y 367.481,Z 546.127,A -85,B 0,C 180,E1 -12696.016,E2 -12696.016} C_VEL
LIN {X 0,Y 367.702,Z 541.891,A -85,B 0,C 180,E1 -12697.692,E2 -12697.692} C_VEL
LIN {X 0,Y 368.129,Z 535.498,A -85,B 0,C 180,E1 -12699.619,E2 -12699.619} C_VEL
LIN {X 0,Y 368.692,Z 528.527,A -85,B 0,C 180,E1 -12701.27,E2 -12701.27} C_VEL
LIN {X 0,Y 369.58,Z 519.787,A -85,B 0,C 180,E1 -12702.914,E2 -12702.914} C_VEL
LIN {X 0,Y 370.516,Z 509.767,A -85,B 0,C 180,E1 -12704.428,E2 -12704.428} C_VEL
LIN {X 0,Y 371.391,Z 499.757,A -85,B 0,C 180,E1 -12705.647,E2 -12705.647} C_VEL
LIN {X 0,Y 372.365,Z 488.548,A -85,B 0,C 180,E1 -12706.73,E2 -12706.73} C_VEL
LIN {X 0,Y 373.359,Z 475.994,A -85,B 0,C 180,E1 -12707.672,E2 -12707.672} C_VEL
LIN {X 0,Y 374.214,Z 463.175,A -85,B 0,C 180,E1 -12708.373,E2 -12708.373} C_VEL
LIN {X 0,Y 374.883,Z 449.6,A -85,B 0,C 180,E1 -12708.87,E2 -12708.87} C_VEL
LIN {X 0,Y 376.193,Z 374.066,A -85,B 0,C 180,E1 -12710.393,E2 -12710.393} C_VEL
LIN {X 0,Y 371.267,Z 340.185,A -85,B 0,C 180,E1 -12711.386,E2 -12711.386} C_VEL
LIN {X 0,Y 372.619,Z 324.581,A -85,B 0,C 180,E1 -12714.833,E2 -12714.833} C_VEL
LIN {X 0,Y 372.299,Z 320.718,A -85,B 0,C 180,E1 -12715.735,E2 -12715.735} C_VEL
LIN {X 0,Y 370.168,Z 310.102,A -85,B 0,C 180,E1 -12718.338,E2 -12718.338} C_VEL
LIN {X 0,Y 368.93,Z 304.531,A -85,B 0,C 180,E1 -12719.769,E2 -12719.769} C_VEL
LIN {X 0,Y 368.902,Z 304.53,A -85,B 0,C 180,E1 -12723.539,E2 -12723.539} C_VEL
LIN {X 0,Y 368.905,Z 304.529,A -85,B 0,C 180,E1 -12726.856,E2 -12726.856} C_VEL
LIN {X 0,Y 368.914,Z 304.534,A -85,B 0,C 180,E1 -12730.371,E2 -12730.371} C_VEL
LIN {X 0,Y 368.885,Z 304.531,A -85,B 0,C 180,E1 -12733.616,E2 -12733.616} C_VEL
LIN {X 0,Y 368.889,Z 304.535,A -85,B 0,C 180,E1 -12736.696,E2 -12736.696} C_VEL
LIN {X 0,Y 368.913,Z 304.527,A -85,B 0,C 180,E1 -12739.644,E2 -12739.644} C_VEL
LIN {X 0,Y 368.902,Z 304.53,A -85,B 0,C 180,E1 -12743.145,E2 -12743.145} C_VEL
LIN {X 0,Y 368.897,Z 304.534,A -85,B 0,C 180,E1 -12746.462,E2 -12746.462} C_VEL
LIN {X 0,Y 368.914,Z 304.529,A -85,B 0,C 180,E1 -12750.31,E2 -12750.31} C_VEL
LIN {X 0,Y 368.999,Z 304.517,A -85,B 0,C 180,E1 -12754.02,E2 -12754.02} C_VEL
LIN {X 0,Y 368.924,Z 304.527,A -85,B 0,C 180,E1 -12757.604,E2 -12757.604} C_VEL
LIN {X 0,Y 368.952,Z 304.529,A -85,B 0,C 180,E1 -12761.106,E2 -12761.106} C_VEL
LIN {X 0,Y 368.993,Z 304.519,A -85,B 0,C 180,E1 -12764.535,E2 -12764.535} C_VEL
LIN {X 0,Y 368.999,Z 304.517,A -85,B 0,C 180,E1 -12767.907,E2 -12767.907} C_VEL
LIN {X 0,Y 369.163,Z 304.497,A -85,B 0,C 180,E1 -12771.87,E2 -12771.87} C_VEL
LIN {X 0,Y 369.134,Z 304.5,A -85,B 0,C 180,E1 -12774.537,E2 -12774.537} C_VEL
LIN {X 0,Y 369.309,Z 304.481,A -85,B 0,C 180,E1 -12777.819,E2 -12777.819} C_VEL
LIN {X 0,Y 369.427,Z 304.465,A -85,B 0,C 180,E1 -12780,E2 -12780} C_VEL
LIN {X 0,Y 369.309,Z 304.479,A -85,B 0,C 180,E1 -12782.181,E2 -12782.181} C_VEL
LIN {X 0,Y 369.156,Z 304.497,A -85,B 0,C 180,E1 -12786.559,E2 -12786.559} C_VEL
LIN {X 0,Y 369.058,Z 304.515,A -85,B 0,C 180,E1 -12789.869,E2 -12789.869} C_VEL
LIN {X 0,Y 369.035,Z 304.519,A -85,B 0,C 180,E1 -12793.772,E2 -12793.772} C_VEL
LIN {X 0,Y 368.99,Z 304.523,A -85,B 0,C 180,E1 -12797.743,E2 -12797.743} C_VEL
LIN {X 0,Y 368.907,Z 304.528,A -85,B 0,C 180,E1 -12801.221,E2 -12801.221} C_VEL
LIN {X 0,Y 368.906,Z 304.533,A -85,B 0,C 180,E1 -12803.873,E2 -12803.873} C_VEL
LIN {X 0,Y 368.856,Z 304.535,A -85,B 0,C 180,E1 -12807.212,E2 -12807.212} C_VEL
LIN {X 0,Y 368.891,Z 304.532,A -85,B 0,C 180,E1 -12809.693,E2 -12809.693} C_VEL
LIN {X 0,Y 368.895,Z 304.53,A -85,B 0,C 180,E1 -12813.538,E2 -12813.538} C_VEL
LIN {X 0,Y 368.894,Z 304.532,A -85,B 0,C 180,E1 -12816.854,E2 -12816.854} C_VEL
LIN {X 0,Y 368.885,Z 304.537,A -85,B 0,C 180,E1 -12820.374,E2 -12820.374} C_VEL
LIN {X 0,Y 368.871,Z 304.533,A -85,B 0,C 180,E1 -12823.613,E2 -12823.613} C_VEL
LIN {X 0,Y 368.848,Z 304.542,A -85,B 0,C 180,E1 -12826.689,E2 -12826.689} C_VEL
LIN {X 0,Y 368.888,Z 304.531,A -85,B 0,C 180,E1 -12829.648,E2 -12829.648} C_VEL
LIN {X 0,Y 368.873,Z 304.535,A -85,B 0,C 180,E1 -12833.15,E2 -12833.15} C_VEL
LIN {X 0,Y 368.866,Z 304.536,A -85,B 0,C 180,E1 -12836.457,E2 -12836.457} C_VEL
LIN {X 0,Y 368.896,Z 304.531,A -85,B 0,C 180,E1 -12840.306,E2 -12840.306} C_VEL
LIN {X 0,Y 368.927,Z 304.526,A -85,B 0,C 180,E1 -12844.012,E2 -12844.012} C_VEL
LIN {X 0,Y 368.903,Z 304.53,A -85,B 0,C 180,E1 -12847.601,E2 -12847.601} C_VEL
LIN {X 0,Y 368.96,Z 304.528,A -85,B 0,C 180,E1 -12851.104,E2 -12851.104} C_VEL
LIN {X 0,Y 369,Z 304.517,A -85,B 0,C 180,E1 -12854.533,E2 -12854.533} C_VEL
LIN {X 0,Y 369.008,Z 304.517,A -85,B 0,C 180,E1 -12857.904,E2 -12857.904} C_VEL
LIN {X 0,Y 369.095,Z 304.51,A -85,B 0,C 180,E1 -12861.235,E2 -12861.235} C_VEL
LIN {X 0,Y 369.119,Z 304.502,A -85,B 0,C 180,E1 -12864.534,E2 -12864.534} C_VEL
LIN {X 0,Y 369.304,Z 304.483,A -85,B 0,C 180,E1 -12867.815,E2 -12867.815} C_VEL
LIN {X 0,Y 369.204,Z 304.492,A -85,B 0,C 180,E1 -12871.087,E2 -12871.087} C_VEL
LIN {X 0,Y 369.304,Z 304.481,A -85,B 0,C 180,E1 -12872.178,E2 -12872.178} C_VEL
LIN {X 0,Y 369.152,Z 304.502,A -85,B 0,C 180,E1 -12876.555,E2 -12876.555} C_VEL
LIN {X 0,Y 369.139,Z 304.585,A -85,B 0,C 180,E1 -12878.017,E2 -12878.017} C_VEL
LIN {X 0,Y 370.937,Z 314.354,A -85,B 0,C 180,E1 -12880.67,E2 -12880.67} C_VEL
LIN {X 0,Y 373.399,Z 322.614,A -85,B 0,C 180,E1 -12880.999,E2 -12880.999} C_VEL
LIN {X 0,Y 376.58,Z 338.412,A -85,B 0,C 180,E1 -12881.501,E2 -12881.501} C_VEL
LIN {X 0,Y 375.113,Z 422.023,A -85,B 0,C 180,E1 -12883.178,E2 -12883.178} C_VEL
LIN {X 0,Y 374.612,Z 435.574,A -85,B 0,C 180,E1 -12883.674,E2 -12883.674} C_VEL
LIN {X 0,Y 373.972,Z 447.98,A -85,B 0,C 180,E1 -12884.345,E2 -12884.345} C_VEL
LIN {X 0,Y 373.257,Z 458.943,A -85,B 0,C 180,E1 -12885.14,E2 -12885.14} C_VEL
LIN {X 0,Y 372.236,Z 471.07,A -85,B 0,C 180,E1 -12886.273,E2 -12886.273} C_VEL
LIN {X 0,Y 371.266,Z 481.361,A -85,B 0,C 180,E1 -12887.483,E2 -12887.483} C_VEL
LIN {X 0,Y 370.478,Z 490.441,A -85,B 0,C 180,E1 -12888.809,E2 -12888.809} C_VEL
LIN {X 0,Y 370.014,Z 494.728,A -85,B 0,C 180,E1 -12889.537,E2 -12889.537} C_VEL
LIN {X 0,Y 369.029,Z 498.529,A -85,B 0,C 180,E1 -12890.228,E2 -12890.228} C_VEL
LIN {X 0,Y 365.694,Z 504.301,A -85,B 0,C 180,E1 -12891.369,E2 -12891.369} C_VEL
LIN {X 0,Y 362.361,Z 509.471,A -85,B 0,C 180,E1 -12892.595,E2 -12892.595} C_VEL
LIN {X 0,Y 361.399,Z 512.236,A -85,B 0,C 180,E1 -12893.409,E2 -12893.409} C_VEL
LIN {X 0,Y 360.909,Z 517.65,A -85,B 0,C 180,E1 -12895.361,E2 -12895.361} C_VEL
LIN {X 0,Y 360.521,Z 521.46,A -85,B 0,C 180,E1 -12897.259,E2 -12897.259} C_VEL
LIN {X 0,Y 360.264,Z 524.038,A -85,B 0,C 180,E1 -12899.183,E2 -12899.183} C_VEL
LIN {X 0,Y 360.178,Z 525.285,A -85,B 0,C 180,E1 -12900.845,E2 -12900.845} C_VEL
LIN {X 0,Y 360.17,Z 525.58,A -85,B 0,C 180,E1 -12903.111,E2 -12903.111} C_VEL
LIN {X 0,Y 360.328,Z 524.563,A -85,B 0,C 180,E1 -12904.996,E2 -12904.996} C_VEL
LIN {X 0,Y 360.633,Z 521.943,A -85,B 0,C 180,E1 -12907.158,E2 -12907.158} C_VEL
LIN {X 0,Y 360.965,Z 518.8,A -85,B 0,C 180,E1 -12908.849,E2 -12908.849} C_VEL
LIN {X 0,Y 361.467,Z 514.159,A -85,B 0,C 180,E1 -12910.687,E2 -12910.687} C_VEL
LIN {X 0,Y 362.158,Z 508.237,A -85,B 0,C 180,E1 -12912.487,E2 -12912.487} C_VEL
LIN {X 0,Y 363.058,Z 500.793,A -85,B 0,C 180,E1 -12914.255,E2 -12914.255} C_VEL
LIN {X 0,Y 364.208,Z 491.511,A -85,B 0,C 180,E1 -12915.998,E2 -12915.998} C_VEL
LIN {X 0,Y 365.29,Z 482.45,A -85,B 0,C 180,E1 -12917.365,E2 -12917.365} C_VEL
LIN {X 0,Y 366.297,Z 472.095,A -85,B 0,C 180,E1 -12918.629,E2 -12918.629} C_VEL
LIN {X 0,Y 367.464,Z 460.727,A -85,B 0,C 180,E1 -12919.725,E2 -12919.725} C_VEL
LIN {X 0,Y 368.365,Z 449.358,A -85,B 0,C 180,E1 -12920.586,E2 -12920.586} C_VEL
LIN {X 0,Y 369.118,Z 436.425,A -85,B 0,C 180,E1 -12921.308,E2 -12921.308} C_VEL
LIN {X 0,Y 369.688,Z 423.36,A -85,B 0,C 180,E1 -12921.8,E2 -12921.8} C_VEL
LIN {X 0,Y 371.403,Z 339.891,A -85,B 0,C 180,E1 -12923.537,E2 -12923.537} C_VEL
LIN {X 0,Y 368.18,Z 325.241,A -85,B 0,C 180,E1 -12924.083,E2 -12924.083} C_VEL
LIN {X 0,Y 363.961,Z 314.71,A -85,B 0,C 180,E1 -12924.641,E2 -12924.641} C_VEL
LIN {X 0,Y 361.833,Z 305.415,A -85,B 0,C 180,E1 -12927.054,E2 -12927.054} C_VEL
LIN {X 0,Y 361.862,Z 305.412,A -85,B 0,C 180,E1 -12930.952,E2 -12930.952} C_VEL
LIN {X 0,Y 361.913,Z 305.409,A -85,B 0,C 180,E1 -12933.472,E2 -12933.472} C_VEL
LIN {X 0,Y 361.844,Z 305.417,A -85,B 0,C 180,E1 -12937.141,E2 -12937.141} C_VEL
LIN {X 0,Y 361.859,Z 305.412,A -85,B 0,C 180,E1 -12940.721,E2 -12940.721} C_VEL
LIN {X 0,Y 361.886,Z 305.406,A -85,B 0,C 180,E1 -12943.064,E2 -12943.064} C_VEL
LIN {X 0,Y 361.952,Z 305.397,A -85,B 0,C 180,E1 -12946.526,E2 -12946.526} C_VEL
LIN {X 0,Y 361.955,Z 305.393,A -85,B 0,C 180,E1 -12949.936,E2 -12949.936} C_VEL
LIN {X 0,Y 362.113,Z 305.377,A -85,B 0,C 180,E1 -12953.313,E2 -12953.313} C_VEL
LIN {X 0,Y 362.234,Z 305.361,A -85,B 0,C 180,E1 -12957.776,E2 -12957.776} C_VEL
LIN {X 0,Y 362.379,Z 305.335,A -85,B 0,C 180,E1 -12960,E2 -12960} C_VEL
LIN {X 0,Y 362.235,Z 305.361,A -85,B 0,C 180,E1 -12962.224,E2 -12962.224} C_VEL
LIN {X 0,Y 362.115,Z 305.378,A -85,B 0,C 180,E1 -12966.687,E2 -12966.687} C_VEL
LIN {X 0,Y 361.989,Z 305.392,A -85,B 0,C 180,E1 -12970.063,E2 -12970.063} C_VEL
LIN {X 0,Y 361.952,Z 305.396,A -85,B 0,C 180,E1 -12973.9,E2 -12973.9} C_VEL
LIN {X 0,Y 361.924,Z 305.398,A -85,B 0,C 180,E1 -12977.941,E2 -12977.941} C_VEL
LIN {X 0,Y 361.882,Z 305.405,A -85,B 0,C 180,E1 -12981.654,E2 -12981.654} C_VEL
LIN {X 0,Y 361.889,Z 305.4,A -85,B 0,C 180,E1 -12985.293,E2 -12985.293} C_VEL
LIN {X 0,Y 361.879,Z 305.4,A -85,B 0,C 180,E1 -12987.782,E2 -12987.782} C_VEL
LIN {X 0,Y 361.809,Z 305.414,A -85,B 0,C 180,E1 -12991.289,E2 -12991.289} C_VEL
